//Error
IF timDissableFunctions.Q THEN 
	fbEM.bWarning := TRUE; 
	fbEM.iWarningCode := 0; 
ELSE 
	fbEM.bWarning := FALSE; 
END_IF 
IF Lynus_Standards.GVL_Energy.stNumberOfDevices.diNumberOfElectricMeters > Constants_Energy.diMaxNumberOfElectricMeters THEN 
	fbEM.bError := TRUE; 
ELSE 
	fbEM.bError := FALSE; 
END_IF
IF Lynus_Standards.GVL_Energy.stNumberOfDevices.diNumberOfElectricMeters > Constants_Energy.diMaxNumberOfElectricMeters THEN 
	fbEM.iErrorCode := 1;
ELSE 
	fbEM.iErrorCode := 0;
END_IF

timSetCounterValues(IN:= bEnable AND NOT timSetCounterValues.Q, PT:= T#2S, Q=> , ET=> );

END_FUNCTION_BLOCK

// ---- FBs/FB_EM_Beckhoff_EL3446.TcPOU
FUNCTION_BLOCK FB_EM_Beckhoff_EL3446
VAR_INPUT
	bEnable							: BOOL;											//Enable the function
  	bEnableVariantValues 			: BOOL; //Enables the Variant values to be queried using the multiplexer functions of the block
    pDpmData 						: POINTER TO ARRAY[1..20] OF UDINT;
	nSlaveAddr						: UINT;											//EtherCat Slave ID	
 	b_SubIndex						: BYTE;											//AmsNet ID Index, typically 2 or 3
 	bInvers_CH1						: BOOL;											//Invert the Output data from Channel 1 
	bInvers_CH2						: BOOL;											//Invert the Output data from Channel 2 
	bInvers_CH3						: BOOL;											//Invert the Output data from Channel 3
	bInvers_CH4						: BOOL;											//Invert the Output data from Channel 4
	bInvers_CH5						: BOOL;											//Invert the Output data from Channel 5
	bInvers_CH6						: BOOL;											//Invert the Output data from Channel 6
	uiCurrentTransformerRatio_CH1	: UINT;											//Current Transformer Ratio for Channel 1 
	uiCurrentTransformerRatio_CH2	: UINT;											//Current Transformer Ratio for Channel 2 
	uiCurrentTransformerRatio_CH3	: UINT;											//Current Transformer Ratio for Channel 3 
	uiCurrentTransformerRatio_CH4	: UINT;											//Current Transformer Ratio for Channel 4 
	uiCurrentTransformerRatio_CH5	: UINT;											//Current Transformer Ratio for Channel 5 
	uiCurrentTransformerRatio_CH6	: UINT;											//Current Transformer Ratio for Channel 6
	uiVoltagePhaseSelector_CH1		: UINT;											//Voltage Phase Selector 1/2/3 for Channel 1
	uiVoltagePhaseSelector_CH2		: UINT;											//Voltage Phase Selector 1/2/3 for Channel 2
	uiVoltagePhaseSelector_CH3		: UINT;											//Voltage Phase Selector 1/2/3 for Channel 3
	uiVoltagePhaseSelector_CH4		: UINT;											//Voltage Phase Selector 1/2/3 for Channel 4
	uiVoltagePhaseSelector_CH5		: UINT;											//Voltage Phase Selector 1/2/3 for Channel 5
	uiVoltagePhaseSelector_CH6		: UINT;											//Voltage Phase Selector 1/2/3 for Channel 6 
	bEnable3PhaseCH13				: BOOL;											//Enable 3 phase measurement Channel 1-3
	bEnable3PhaseCH46				: BOOL;											//Enable 3 phase measurement Channel 4-6
	stDataEMPowerRealTime			: ST_ElectricMeter_Output_Power;				//Output structure with Data from Electric Meter (Power Data RealTime) used adding voltage to output struct
    stEL3446_IO : MDP5001_342_066CA8C6; 
END_VAR
VAR_OUTPUT
	stDataEMPower_CH1				: ST_ElectricMeter_Output_Power;				//Output structure with Data from Electric Meter (Power Data) for Channel 1
	stDataEMCounter_CH1				: ST_ElectricMeter_Output_Counter;				//Output structure with Data from Electric Meter (Counter Data) for Channel 1
	stDataEMPowerRealTime_CH1		: ST_ElectricMeter_Output_Power;				//Output structure with Data from Electric Meter (Power Data RealTime) for Channel 1
	stDataEMCounterRealTime_CH1		: ST_ElectricMeter_Output_Counter;				//Output structure with Data from Electric Meter (Counter Data RealTime) for Channel 1

	stDataEMPower_CH2				: ST_ElectricMeter_Output_Power;				//Output structure with Data from Electric Meter (Power Data) for Channel 2
	stDataEMCounter_CH2				: ST_ElectricMeter_Output_Counter;				//Output structure with Data from Electric Meter (Counter Data) for Channel 2
	stDataEMPowerRealTime_CH2		: ST_ElectricMeter_Output_Power;				//Output structure with Data from Electric Meter (Power Data RealTime) for Channel 2
	stDataEMCounterRealTime_CH2		: ST_ElectricMeter_Output_Counter;				//Output structure with Data from Electric Meter (Counter Data RealTime) for Channel 2

	stDataEMPower_CH3				: ST_ElectricMeter_Output_Power;				//Output structure with Data from Electric Meter (Power Data) for Channel 3
	stDataEMCounter_CH3				: ST_ElectricMeter_Output_Counter;				//Output structure with Data from Electric Meter (Counter Data) for Channel 3
	stDataEMPowerRealTime_CH3		: ST_ElectricMeter_Output_Power;				//Output structure with Data from Electric Meter (Power Data RealTime) for Channel 3
	stDataEMCounterRealTime_CH3		: ST_ElectricMeter_Output_Counter;				//Output structure with Data from Electric Meter (Counter Data RealTime) for Channel 3

	stDataEMPower_CH4				: ST_ElectricMeter_Output_Power;				//Output structure with Data from Electric Meter (Power Data) for Channel 4
	stDataEMCounter_CH4				: ST_ElectricMeter_Output_Counter;				//Output structure with Data from Electric Meter (Counter Data) for Channel 4
	stDataEMPowerRealTime_CH4		: ST_ElectricMeter_Output_Power;				//Output structure with Data from Electric Meter (Power Data RealTime) for Channel 4
	stDataEMCounterRealTime_CH4		: ST_ElectricMeter_Output_Counter;				//Output structure with Data from Electric Meter (Counter Data RealTime) for Channel 4

	stDataEMPower_CH5				: ST_ElectricMeter_Output_Power;				//Output structure with Data from Electric Meter (Power Data) for Channel 5
	stDataEMCounter_CH5				: ST_ElectricMeter_Output_Counter;				//Output structure with Data from Electric Meter (Counter Data) for Channel 5
	stDataEMPowerRealTime_CH5		: ST_ElectricMeter_Output_Power;				//Output structure with Data from Electric Meter (Power Data RealTime) for Channel 5
	stDataEMCounterRealTime_CH5		: ST_ElectricMeter_Output_Counter;				//Output structure with Data from Electric Meter (Counter Data RealTime) for Channel 5

	stDataEMPower_CH6				: ST_ElectricMeter_Output_Power;				//Output structure with Data from Electric Meter (Power Data) for Channel 6
	stDataEMCounter_CH6				: ST_ElectricMeter_Output_Counter;				//Output structure with Data from Electric Meter (Counter Data) for Channel 6
	stDataEMPowerRealTime_CH6		: ST_ElectricMeter_Output_Power;				//Output structure with Data from Electric Meter (Power Data RealTime) for Channel 6
	stDataEMCounterRealTime_CH6		: ST_ElectricMeter_Output_Counter;				//Output structure with Data from Electric Meter (Counter Data RealTime) for Channel 6	
	
END_VAR
VAR
	fbEM_CH1						: FB_ElectricMeter;								//Electric Meter Function
	fbEnergyCounter_CH1				: FB_EnergyCounter;								//FB energy Counter, because the KL3403 has no nice logic for the Energy value
	fbEM_CH2						: FB_ElectricMeter;								//Electric Meter Function
	fbEnergyCounter_CH2				: FB_EnergyCounter;								//FB energy Counter, because the KL3403 has no nice logic for the Energy value
	fbEM_CH3						: FB_ElectricMeter;								//Electric Meter Function
	fbEnergyCounter_CH3				: FB_EnergyCounter;								//FB energy Counter, because the KL3403 has no nice logic for the Energy value
	fbEM_CH4						: FB_ElectricMeter;								//Electric Meter Function
	fbEnergyCounter_CH4				: FB_EnergyCounter;								//FB energy Counter, because the KL3403 has no nice logic for the Energy value
	fbEM_CH5						: FB_ElectricMeter;								//Electric Meter Function
	fbEnergyCounter_CH5				: FB_EnergyCounter;								//FB energy Counter, because the KL3403 has no nice logic for the Energy value
	fbEM_CH6						: FB_ElectricMeter;								//Electric Meter Function
	fbEnergyCounter_CH6				: FB_EnergyCounter;								//FB energy Counter, because the KL3403 has no nice logic for the Energy value
	fbEL3446_wEL3443	: FB_EL3446; 		//EL3446 | 6-channel current input terminal 1 A AC/DC for distributed power measurement (FW02 or higher) for DPM with EL3443
	
	timDissableFunctions			: TON;											//Timer to dissable the Function after Lynus_Standards.Constants_General.tTimeDissableLynusFunctions Days without connection to the Lynus Cloud
	timResetConnectionOnGVL			: TON;											//Timer to try reset the connection Flag on the GVL. (When somebody delete the Connection Function and make only a onlinechange)
	timSetCounterValues				: TON;											//Timer to set the counter values from the KL3403 Function to the EM Function
	arrPD							: ARRAY[1..7] OF FB_PersistentData_Number;		//Function to save persistent data
	byWaitInStep					: BYTE;											//Wait in Step before start to clean data on PLC
	iStateGVLData					: INT;											//State machine to handle the data on the GVL
	diCounterForGVL					: DINT;											//Counter to clean old data on GVL
	bInit: BOOL;
	m_COE_Done: BOOL;
	FB_CoE_EL3446 :FB_CoE_EL3446;
	uiVoltagePhaseSelector_old_CH1		: UINT;											
	uiVoltagePhaseSelector_old_CH2		: UINT;											
	uiVoltagePhaseSelector_old_CH3		: UINT;											
	uiVoltagePhaseSelector_old_CH4		: UINT;											
	uiVoltagePhaseSelector_old_CH5		: UINT;											
	uiVoltagePhaseSelector_old_CH6		: UINT;											
	
	f_trig_Busy: f_trig;

	real_Multiplier_CH1: REAL;
	real_Multiplier_CH2: REAL;
	real_Multiplier_CH3: REAL;
	real_Multiplier_CH4: REAL;
	real_Multiplier_CH5: REAL;
	real_Multiplier_CH6: REAL;
	

			
END_VAR

//Creator : Stefan Lackner
//Company : EfficientIO
//Date : xx.09.2023
//Version : 1.0.0.0


//With this function is possible to read out all Information from a EL3446

//NOTE for diNr.....Designation => 
//_IN = Here Data come in from other Functions or go out to other functions about the GVL
//_OUT = Here Data go out to other functions about the GVL



(*-------------------------------------------------------------Service from Backend is ready and check the connection to backen for dissabel/enable Function---------------------------------------------------------------*)

//Try to reset the variable for connection on the GVL. When all is normal then the Lynus Mqtt connection function set this variable to true in the next cycle
//When we have no connection to the backend then after Lynus_Standards.Constants_General.tTimeDissableLynusFunctions days the Function is dissabled with all of his functionalities
timResetConnectionOnGVL(IN:= NOT timResetConnectionOnGVL.Q, PT:= T#1H, Q=> , ET=> );
IF timResetConnectionOnGVL.Q THEN 
	Lynus_Standards.GVL_Communicator.bStateConnectionToEnableFunctions := FALSE; 
END_IF
IF NOT Lynus_Standards.GVL_Communicator.bStateConnectionToEnableFunctions THEN 
	timDissableFunctions.IN := TRUE; 
ELSE 
	timDissableFunctions.IN := FALSE; 
END_IF  
timDissableFunctions(IN:= , PT:= Lynus_Standards.Constants_General.tTimeDissableLynusFunctions, Q=> , ET=> );

// limit inputs
uiCurrentTransformerRatio_CH1 := LIMIT (1,uiCurrentTransformerRatio_CH1,10000);
uiCurrentTransformerRatio_CH2 := LIMIT (1,uiCurrentTransformerRatio_CH2,10000);
uiCurrentTransformerRatio_CH3 := LIMIT (1,uiCurrentTransformerRatio_CH3,10000);
uiCurrentTransformerRatio_CH4 := LIMIT (1,uiCurrentTransformerRatio_CH4,10000);
uiCurrentTransformerRatio_CH5 := LIMIT (1,uiCurrentTransformerRatio_CH5,10000);
uiCurrentTransformerRatio_CH6 := LIMIT (1,uiCurrentTransformerRatio_CH6,10000);
uiVoltagePhaseSelector_CH1 := LIMIT (1,uiVoltagePhaseSelector_CH1,3);
uiVoltagePhaseSelector_CH2 := LIMIT (1,uiVoltagePhaseSelector_CH2,3);
uiVoltagePhaseSelector_CH3 := LIMIT (1,uiVoltagePhaseSelector_CH3,3);
uiVoltagePhaseSelector_CH4 := LIMIT (1,uiVoltagePhaseSelector_CH4,3);
uiVoltagePhaseSelector_CH5 := LIMIT (1,uiVoltagePhaseSelector_CH5,3);
uiVoltagePhaseSelector_CH6 := LIMIT (1,uiVoltagePhaseSelector_CH6,3);


(*----------------------------------------------------------------------------------------EL3446 Communication----------------------------------------------------------------------------------------------*)

// write CoE values for phase selector

IF 	NOT m_COE_Done OR uiVoltagePhaseSelector_CH1 <> uiVoltagePhaseSelector_old_CH1 OR uiVoltagePhaseSelector_CH2 <> uiVoltagePhaseSelector_old_CH2 OR
 	uiVoltagePhaseSelector_CH3 <> uiVoltagePhaseSelector_old_CH3 OR uiVoltagePhaseSelector_CH4 <> uiVoltagePhaseSelector_old_CH4 OR
  	uiVoltagePhaseSelector_CH5 <> uiVoltagePhaseSelector_old_CH5 OR uiVoltagePhaseSelector_CH6 <> uiVoltagePhaseSelector_old_CH6 
	THEN
	FB_CoE_EL3446.m_start := TRUE;
	m_COE_Done := TRUE;
	 uiVoltagePhaseSelector_old_CH1 := uiVoltagePhaseSelector_CH1;
	 uiVoltagePhaseSelector_old_CH2 := uiVoltagePhaseSelector_CH2;
	 uiVoltagePhaseSelector_old_CH3 := uiVoltagePhaseSelector_CH3;
	 uiVoltagePhaseSelector_old_CH4 := uiVoltagePhaseSelector_CH4;
	 uiVoltagePhaseSelector_old_CH5 := uiVoltagePhaseSelector_CH5;
	 uiVoltagePhaseSelector_old_CH6 := uiVoltagePhaseSelector_CH6;
END_IF
f_trig_Busy(CLK := FB_CoE_EL3446.m_Busy );
IF f_trig_Busy.Q AND (FB_CoE_EL3446.m_CoE_Write_done OR FB_CoE_EL3446.m_Error) THEN 
	FB_CoE_EL3446.m_start := FALSE;
END_IF
FB_CoE_EL3446(
	m_start:= , 
	nSlaveAddr:= nSlaveAddr,
	b_SubIndex:= b_SubIndex,
	uiVoltagePhaseSelector_CH1:= uiVoltagePhaseSelector_CH1, 
	uiVoltagePhaseSelector_CH2:= uiVoltagePhaseSelector_CH2, 
	uiVoltagePhaseSelector_CH3:= uiVoltagePhaseSelector_CH3, 
	uiVoltagePhaseSelector_CH4:= uiVoltagePhaseSelector_CH4, 
	uiVoltagePhaseSelector_CH5:= uiVoltagePhaseSelector_CH5, 
	uiVoltagePhaseSelector_CH6:= uiVoltagePhaseSelector_CH6, 
	m_Busy=> , 
	m_CoE_Write_done=> , 
	udint_GetAMSNetID_Error=> , 
	udint_WriteCoE_Error=> );

fbEL3446_wEL3443(
	bEnable:= TRUE, 
	pDpmData:= pDpmData, 
	stEL3446_IO:= , 
	stStatusPhase_I1=> , 
	stStatusPhase_I2=> , 
	stStatusPhase_I3=> , 
	stStatusPhase_I4=> , 
	stStatusPhase_I5=> , 
	stStatusPhase_I6=> , 
	stDPMVariantValues=> , 
	bError=> );
fbEL3446_wEL3443.stEL3446_IO.MDP5001_342_Input := stEL3446_IO.MDP5001_342_Input;
stEL3446_IO.MDP5001_342_Output := fbEL3446_wEL3443.stEL3446_IO.MDP5001_342_Output;
//Invert the Output data, because it is possible that the current transformers have been mounted in different mounting positions.
IF NOT bInvers_CH1 THEN
	real_Multiplier_CH1 := 1;
ELSE
	real_Multiplier_CH1 := -1;
END_IF
IF NOT bInvers_CH2 THEN
	real_Multiplier_CH2 := 1;
ELSE
	real_Multiplier_CH2 := -1;
END_IF
IF NOT bInvers_CH3 THEN
	real_Multiplier_CH3 := 1;
ELSE
	real_Multiplier_CH3 := -1;
END_IF
IF NOT bInvers_CH4 THEN
	real_Multiplier_CH4 := 1;
ELSE
	real_Multiplier_CH4 := -1;
END_IF
IF NOT bInvers_CH5 THEN
	real_Multiplier_CH5 := 1;
ELSE
	real_Multiplier_CH5 := -1;
END_IF
IF NOT bInvers_CH6 THEN
	real_Multiplier_CH6 := 1;
ELSE
	real_Multiplier_CH6 := -1;
END_IF

//Function
IF NOT bEnable3PhaseCH13 THEN
	fbEM_CH1(
		bEnable:= bEnable AND NOT timDissableFunctions.Q, 
		bError:= , 
		bEnableReadOutFunction:= FALSE, 
		bWriteWithDelay:= TRUE, 
		bPowerDataInvers:= FALSE,
		bReadOutDataDone:= timSetCounterValues.Q,
		iTimeReadOutInterval:= 0, 
		iErrorCode:= , 
		iWarningCode:= , 
		lrTotalCounterEnergy_Consumption:= fbEnergyCounter_CH1.lrTotalCounterEnergy_Consumption,
		lrTotalCounterEnergy_Production:= fbEnergyCounter_CH1.lrTotalCounterEnergy_Production, 
		lrCounterEnergyT1_Consumption:= fbEnergyCounter_CH1.lrCounterEnergyT1_Consumption,
		lrCounterEnergyT2_Consumption:= fbEnergyCounter_CH1.lrCounterEnergyT2_Consumption,
		lrCounterEnergyT1_Production:= fbEnergyCounter_CH1.lrCounterEnergyT1_Production, 
		lrCounterEnergyT2_Production:= fbEnergyCounter_CH1.lrCounterEnergyT2_Production, 
		lrCurrentL1:=  fbEL3446_wEL3443.stStatusPhase_I1.fCurrent * uiCurrentTransformerRatio_CH1,
		lrVoltageL1N:= , 
		lrVoltageL1L2:= , 
		lrPowerL1:= fbEL3446_wEL3443.stStatusPhase_I1.fActive_Power * uiCurrentTransformerRatio_CH1 * real_Multiplier_CH1, 
		lrCurrentL2:= ,
		lrVoltageL2N:= , 
		lrVoltageL2L3:= , 
		lrPowerL2:= , 
		lrCurrentL3:= , 
		lrVoltageL3N:= , 
		lrVoltageL3L1:= , 
		lrPowerL3:= , 
		lrPowerTotal:= fbEM_CH1.lrPowerL1, 
		lrFrequency:= stDataEMPowerRealTime.lrFrequency,  
		lrApparentPowerTotal:= fbEL3446_wEL3443.stStatusPhase_I1.fApparent_Power * uiCurrentTransformerRatio_CH1 ,
		lrReactivePowerTotal:= fbEL3446_wEL3443.stStatusPhase_I1.fReactive_Power_Fundamental * uiCurrentTransformerRatio_CH1, 
		tTimDelayOutput:= T#5S, 
		stDataEMOutPower=> stDataEMPowerRealTime_CH1, 
		stDataEMOutPowerDelay=> stDataEMPower_CH1, 
		stDataEMOutCounter=> stDataEMCounterRealTime_CH1,
		stDataEMOutCounterDelay=> stDataEMCounter_CH1,
		bReadOutMeter=> );
	fbEM_CH2(
		bEnable:= bEnable AND NOT timDissableFunctions.Q, 
		bError:= , 
		bEnableReadOutFunction:= FALSE, 
		bWriteWithDelay:= TRUE, 
		bPowerDataInvers:= FALSE,
		bReadOutDataDone:= timSetCounterValues.Q,
		iTimeReadOutInterval:= 0, 
		iErrorCode:= , 
		iWarningCode:= , 
		lrTotalCounterEnergy_Consumption:= fbEnergyCounter_CH2.lrTotalCounterEnergy_Consumption,
		lrTotalCounterEnergy_Production:= fbEnergyCounter_CH2.lrTotalCounterEnergy_Production, 
		lrCounterEnergyT1_Consumption:= fbEnergyCounter_CH2.lrCounterEnergyT1_Consumption,
		lrCounterEnergyT2_Consumption:= fbEnergyCounter_CH2.lrCounterEnergyT2_Consumption,
		lrCounterEnergyT1_Production:= fbEnergyCounter_CH2.lrCounterEnergyT1_Production, 
		lrCounterEnergyT2_Production:= fbEnergyCounter_CH2.lrCounterEnergyT2_Production, 
		lrCurrentL1:=  fbEL3446_wEL3443.stStatusPhase_I2.fCurrent * uiCurrentTransformerRatio_CH2,
		lrVoltageL1N:= , 
		lrVoltageL1L2:= , 
		lrPowerL1:= fbEL3446_wEL3443.stStatusPhase_I2.fActive_Power * uiCurrentTransformerRatio_CH2 * real_Multiplier_CH2, 
		lrCurrentL2:= ,
		lrVoltageL2N:= , 
		lrVoltageL2L3:= , 
		lrPowerL2:= , 
		lrCurrentL3:= , 
		lrVoltageL3N:= , 
		lrVoltageL3L1:= , 
		lrPowerL3:= , 
		lrPowerTotal:= fbEM_CH2.lrPowerL1, 
		lrFrequency:= stDataEMPowerRealTime.lrFrequency, 
		lrApparentPowerTotal:= fbEL3446_wEL3443.stStatusPhase_I2.fApparent_Power * uiCurrentTransformerRatio_CH2 ,
		lrReactivePowerTotal:= fbEL3446_wEL3443.stStatusPhase_I2.fReactive_Power_Fundamental * uiCurrentTransformerRatio_CH2, 
		tTimDelayOutput:= T#5S, 
		stDataEMOutPower=> stDataEMPowerRealTime_CH2, 
		stDataEMOutPowerDelay=> stDataEMPower_CH2, 
		stDataEMOutCounter=> stDataEMCounterRealTime_CH2,
		stDataEMOutCounterDelay=> stDataEMCounter_CH2,
		bReadOutMeter=> );
	fbEM_CH3(
		bEnable:= bEnable AND NOT timDissableFunctions.Q, 
		bError:= , 
		bEnableReadOutFunction:= FALSE, 
		bWriteWithDelay:= TRUE, 
		bPowerDataInvers:= FALSE,
		bReadOutDataDone:= timSetCounterValues.Q,
		iTimeReadOutInterval:= 0, 
		iErrorCode:= , 
		iWarningCode:= , 
		lrTotalCounterEnergy_Consumption:= fbEnergyCounter_CH3.lrTotalCounterEnergy_Consumption,
		lrTotalCounterEnergy_Production:= fbEnergyCounter_CH3.lrTotalCounterEnergy_Production, 
		lrCounterEnergyT1_Consumption:= fbEnergyCounter_CH3.lrCounterEnergyT1_Consumption,
		lrCounterEnergyT2_Consumption:= fbEnergyCounter_CH3.lrCounterEnergyT2_Consumption,
		lrCounterEnergyT1_Production:= fbEnergyCounter_CH3.lrCounterEnergyT1_Production, 
		lrCounterEnergyT2_Production:= fbEnergyCounter_CH3.lrCounterEnergyT2_Production, 
		lrCurrentL1:=  fbEL3446_wEL3443.stStatusPhase_I3.fCurrent * uiCurrentTransformerRatio_CH3,
		lrVoltageL1N:= , 
		lrVoltageL1L2:= , 
		lrPowerL1:= fbEL3446_wEL3443.stStatusPhase_I3.fActive_Power * uiCurrentTransformerRatio_CH3 * real_Multiplier_CH3, 
		lrCurrentL2:= ,
		lrVoltageL2N:= , 
		lrVoltageL2L3:= , 
		lrPowerL2:= , 
		lrCurrentL3:= , 
		lrVoltageL3N:= , 
		lrVoltageL3L1:= , 
		lrPowerL3:= , 
		lrPowerTotal:= fbEM_CH3.lrPowerL1, 
		lrFrequency:= stDataEMPowerRealTime.lrFrequency,
		lrApparentPowerTotal:= fbEL3446_wEL3443.stStatusPhase_I3.fApparent_Power * uiCurrentTransformerRatio_CH3 ,
		lrReactivePowerTotal:= fbEL3446_wEL3443.stStatusPhase_I3.fReactive_Power_Fundamental * uiCurrentTransformerRatio_CH3, 
		tTimDelayOutput:= T#5S, 
		stDataEMOutPower=> stDataEMPowerRealTime_CH3, 
		stDataEMOutPowerDelay=> stDataEMPower_CH3, 
		stDataEMOutCounter=> stDataEMCounterRealTime_CH3,
		stDataEMOutCounterDelay=> stDataEMCounter_CH3,
		bReadOutMeter=> );
	fbEnergyCounter_CH1(
		byActiveTariff:= 1, 
		lrPowerInput:= (fbEM_CH1.lrPowerL1) / 1000, 
		lrTotalCounterEnergy_Consumption=> , 
		lrTotalCounterEnergy_Production=> , 
		lrCounterEnergyT1_Consumption=> , 
		lrCounterEnergyT2_Consumption=> , 
		lrCounterEnergyT1_Production=> , 
		lrCounterEnergyT2_Production=> );
	fbEnergyCounter_CH2(
		byActiveTariff:= 1, 
		lrPowerInput:= (fbEM_CH2.lrPowerL1) / 1000, 
		lrTotalCounterEnergy_Consumption=> , 
		lrTotalCounterEnergy_Production=> , 
		lrCounterEnergyT1_Consumption=> , 
		lrCounterEnergyT2_Consumption=> , 
		lrCounterEnergyT1_Production=> , 
		lrCounterEnergyT2_Production=> );
	fbEnergyCounter_CH3(
		byActiveTariff:= 1, 
		lrPowerInput:= (fbEM_CH3.lrPowerL1) / 1000, 
		lrTotalCounterEnergy_Consumption=> , 
		lrTotalCounterEnergy_Production=> , 
		lrCounterEnergyT1_Consumption=> , 
		lrCounterEnergyT2_Consumption=> , 
		lrCounterEnergyT1_Production=> , 
		lrCounterEnergyT2_Production=> );
	CASE uiVoltagePhaseSelector_CH1 OF
		1: 	fbEM_CH1.lrVoltageL1N := stDataEMPowerRealTime.lrVoltageL1N;
		2: 	fbEM_CH1.lrVoltageL1N := stDataEMPowerRealTime.lrVoltageL2N;
		3: 	fbEM_CH1.lrVoltageL1N := stDataEMPowerRealTime.lrVoltageL3N;	
	END_CASE
	CASE uiVoltagePhaseSelector_CH2 OF
		1: 	fbEM_CH2.lrVoltageL1N := stDataEMPowerRealTime.lrVoltageL1N;
		2: 	fbEM_CH2.lrVoltageL1N := stDataEMPowerRealTime.lrVoltageL2N;
		3: 	fbEM_CH2.lrVoltageL1N := stDataEMPowerRealTime.lrVoltageL3N;	
	END_CASE
	CASE uiVoltagePhaseSelector_CH3 OF
		1: 	fbEM_CH3.lrVoltageL1N := stDataEMPowerRealTime.lrVoltageL1N;
		2: 	fbEM_CH3.lrVoltageL1N := stDataEMPowerRealTime.lrVoltageL2N;
		3: 	fbEM_CH3.lrVoltageL1N := stDataEMPowerRealTime.lrVoltageL3N;	
	END_CASE	
ELSE
	fbEM_CH1(
		bEnable:= bEnable AND NOT timDissableFunctions.Q, 
		bError:= , 
		bEnableReadOutFunction:= FALSE, 
		bWriteWithDelay:= TRUE, 
		bPowerDataInvers:= FALSE,
		bReadOutDataDone:= timSetCounterValues.Q,
		iTimeReadOutInterval:= 0, 
		iErrorCode:= , 
		iWarningCode:= , 
		lrTotalCounterEnergy_Consumption:= fbEnergyCounter_CH1.lrTotalCounterEnergy_Consumption,
		lrTotalCounterEnergy_Production:= fbEnergyCounter_CH1.lrTotalCounterEnergy_Production, 
		lrCounterEnergyT1_Consumption:= fbEnergyCounter_CH1.lrCounterEnergyT1_Consumption,
		lrCounterEnergyT2_Consumption:= fbEnergyCounter_CH1.lrCounterEnergyT2_Consumption,
		lrCounterEnergyT1_Production:= fbEnergyCounter_CH1.lrCounterEnergyT1_Production, 
		lrCounterEnergyT2_Production:= fbEnergyCounter_CH1.lrCounterEnergyT2_Production, 
		lrCurrentL1:=  fbEL3446_wEL3443.stStatusPhase_I1.fCurrent * uiCurrentTransformerRatio_CH1,
		lrVoltageL1N:= stDataEMPowerRealTime.lrVoltageL1N, 
		lrVoltageL1L2:= stDataEMPowerRealTime.lrVoltageL1L2, 
		lrPowerL1:= fbEL3446_wEL3443.stStatusPhase_I1.fActive_Power * uiCurrentTransformerRatio_CH1 * real_Multiplier_CH1, 
		lrCurrentL2:= fbEL3446_wEL3443.stStatusPhase_I2.fCurrent * uiCurrentTransformerRatio_CH2,
		lrVoltageL2N:= stDataEMPowerRealTime.lrVoltageL2N, 
		lrVoltageL2L3:=stDataEMPowerRealTime.lrVoltageL2L3 , 
		lrPowerL2:= fbEL3446_wEL3443.stStatusPhase_I2.fActive_Power * uiCurrentTransformerRatio_CH2 * real_Multiplier_CH2, 
		lrCurrentL3:=  fbEL3446_wEL3443.stStatusPhase_I3.fCurrent * uiCurrentTransformerRatio_CH3, 
		lrVoltageL3N:= stDataEMPowerRealTime.lrVoltageL3N, 
		lrVoltageL3L1:= stDataEMPowerRealTime.lrVoltageL3L1 , 
		lrPowerL3:= fbEL3446_wEL3443.stStatusPhase_I3.fActive_Power * uiCurrentTransformerRatio_CH3 * real_Multiplier_CH3, 
		lrPowerTotal:= fbEM_CH1.lrPowerL1 + fbEM_CH1.lrPowerL2 + fbEM_CH1.lrPowerL3,
		lrFrequency:= stDataEMPowerRealTime.lrFrequency, 
		lrApparentPowerTotal:= fbEL3446_wEL3443.stStatusPhase_I1.fApparent_Power * uiCurrentTransformerRatio_CH1 + fbEL3446_wEL3443.stStatusPhase_I2.fApparent_Power * uiCurrentTransformerRatio_CH2 + fbEL3446_wEL3443.stStatusPhase_I3.fApparent_Power * uiCurrentTransformerRatio_CH3,
		lrReactivePowerTotal:= fbEL3446_wEL3443.stStatusPhase_I1.fReactive_Power_Fundamental * uiCurrentTransformerRatio_CH1 + fbEL3446_wEL3443.stStatusPhase_I2.fReactive_Power_Fundamental * uiCurrentTransformerRatio_CH2 + fbEL3446_wEL3443.stStatusPhase_I3.fReactive_Power_Fundamental * uiCurrentTransformerRatio_CH3, 
		tTimDelayOutput:= T#5S, 
		stDataEMOutPower=> stDataEMPowerRealTime_CH1, 
		stDataEMOutPowerDelay=> stDataEMPower_CH1, 
		stDataEMOutCounter=> stDataEMCounterRealTime_CH1,
		stDataEMOutCounterDelay=> stDataEMCounter_CH1,
		bReadOutMeter=> );	
	fbEnergyCounter_CH1(
		byActiveTariff:= 1, 
		lrPowerInput:= (fbEM_CH1.lrPowerTotal) / 1000, 
		lrTotalCounterEnergy_Consumption=> , 
		lrTotalCounterEnergy_Production=> , 
		lrCounterEnergyT1_Consumption=> , 
		lrCounterEnergyT2_Consumption=> , 
		lrCounterEnergyT1_Production=> , 
		lrCounterEnergyT2_Production=> );
END_IF	
IF NOT bEnable3PhaseCH46 THEN 	
	fbEM_CH4(
		bEnable:= bEnable AND NOT timDissableFunctions.Q, 
		bError:= , 
		bEnableReadOutFunction:= FALSE, 
		bWriteWithDelay:= TRUE, 
		bPowerDataInvers:= FALSE,
		bReadOutDataDone:= timSetCounterValues.Q,
		iTimeReadOutInterval:= 0, 
		iErrorCode:= , 
		iWarningCode:= , 
		lrTotalCounterEnergy_Consumption:= fbEnergyCounter_CH4.lrTotalCounterEnergy_Consumption,
		lrTotalCounterEnergy_Production:= fbEnergyCounter_CH4.lrTotalCounterEnergy_Production, 
		lrCounterEnergyT1_Consumption:= fbEnergyCounter_CH4.lrCounterEnergyT1_Consumption,
		lrCounterEnergyT2_Consumption:= fbEnergyCounter_CH4.lrCounterEnergyT2_Consumption,
		lrCounterEnergyT1_Production:= fbEnergyCounter_CH4.lrCounterEnergyT1_Production, 
		lrCounterEnergyT2_Production:= fbEnergyCounter_CH4.lrCounterEnergyT2_Production, 
		lrCurrentL1:=  fbEL3446_wEL3443.stStatusPhase_I4.fCurrent * uiCurrentTransformerRatio_CH4,
		lrVoltageL1N:= , 
		lrVoltageL1L2:= , 
		lrPowerL1:= fbEL3446_wEL3443.stStatusPhase_I4.fActive_Power * uiCurrentTransformerRatio_CH4 * real_Multiplier_CH4, 
		lrCurrentL2:= ,
		lrVoltageL2N:= , 
		lrVoltageL2L3:= , 
		lrPowerL2:= , 
		lrCurrentL3:= , 
		lrVoltageL3N:= , 
		lrVoltageL3L1:= , 
		lrPowerL3:= , 
		lrPowerTotal:= fbEM_CH4.lrPowerL1, 
		lrFrequency:= stDataEMPowerRealTime.lrFrequency,
		lrApparentPowerTotal:= fbEL3446_wEL3443.stStatusPhase_I4.fApparent_Power * uiCurrentTransformerRatio_CH4 ,
		lrReactivePowerTotal:= fbEL3446_wEL3443.stStatusPhase_I4.fReactive_Power_Fundamental * uiCurrentTransformerRatio_CH4, 
		tTimDelayOutput:= T#5S, 
		stDataEMOutPower=> stDataEMPowerRealTime_CH4, 
		stDataEMOutPowerDelay=> stDataEMPower_CH4, 
		stDataEMOutCounter=> stDataEMCounterRealTime_CH4,
		stDataEMOutCounterDelay=> stDataEMCounter_CH4,
		bReadOutMeter=> );
	fbEM_CH5(
		bEnable:= bEnable AND NOT timDissableFunctions.Q, 
		bError:= , 
		bEnableReadOutFunction:= FALSE, 
		bWriteWithDelay:= TRUE, 
		bPowerDataInvers:= FALSE,
		bReadOutDataDone:= timSetCounterValues.Q,
		iTimeReadOutInterval:= 0, 
		iErrorCode:= , 
		iWarningCode:= , 
		lrTotalCounterEnergy_Consumption:= fbEnergyCounter_CH5.lrTotalCounterEnergy_Consumption,
		lrTotalCounterEnergy_Production:= fbEnergyCounter_CH5.lrTotalCounterEnergy_Production, 
		lrCounterEnergyT1_Consumption:= fbEnergyCounter_CH5.lrCounterEnergyT1_Consumption,
		lrCounterEnergyT2_Consumption:= fbEnergyCounter_CH5.lrCounterEnergyT2_Consumption,
		lrCounterEnergyT1_Production:= fbEnergyCounter_CH5.lrCounterEnergyT1_Production, 
		lrCounterEnergyT2_Production:= fbEnergyCounter_CH5.lrCounterEnergyT2_Production, 
		lrCurrentL1:=  fbEL3446_wEL3443.stStatusPhase_I5.fCurrent * uiCurrentTransformerRatio_CH5,
		lrVoltageL1N:= , 
		lrVoltageL1L2:= , 
		lrPowerL1:= fbEL3446_wEL3443.stStatusPhase_I5.fActive_Power * uiCurrentTransformerRatio_CH5 * real_Multiplier_CH5, 
		lrCurrentL2:= ,
		lrVoltageL2N:= , 
		lrVoltageL2L3:= , 
		lrPowerL2:= , 
		lrCurrentL3:= , 
		lrVoltageL3N:= , 
		lrVoltageL3L1:= , 
		lrPowerL3:= , 
		lrPowerTotal:= fbEM_CH5.lrPowerL1, 
		lrFrequency:= stDataEMPowerRealTime.lrFrequency,
		lrApparentPowerTotal:= fbEL3446_wEL3443.stStatusPhase_I5.fApparent_Power * uiCurrentTransformerRatio_CH5 ,
		lrReactivePowerTotal:= fbEL3446_wEL3443.stStatusPhase_I5.fReactive_Power_Fundamental * uiCurrentTransformerRatio_CH5, 
		tTimDelayOutput:= T#5S, 
		stDataEMOutPower=> stDataEMPowerRealTime_CH5, 
		stDataEMOutPowerDelay=> stDataEMPower_CH5, 
		stDataEMOutCounter=> stDataEMCounterRealTime_CH5,
		stDataEMOutCounterDelay=> stDataEMCounter_CH5,
		bReadOutMeter=> );
	fbEM_CH6(
		bEnable:= bEnable AND NOT timDissableFunctions.Q, 
		bError:= , 
		bEnableReadOutFunction:= FALSE, 
		bWriteWithDelay:= TRUE, 
		bPowerDataInvers:= FALSE,
		bReadOutDataDone:= timSetCounterValues.Q,
		iTimeReadOutInterval:= 0, 
		iErrorCode:= , 
		iWarningCode:= , 
		lrTotalCounterEnergy_Consumption:= fbEnergyCounter_CH6.lrTotalCounterEnergy_Consumption,
		lrTotalCounterEnergy_Production:= fbEnergyCounter_CH6.lrTotalCounterEnergy_Production, 
		lrCounterEnergyT1_Consumption:= fbEnergyCounter_CH6.lrCounterEnergyT1_Consumption,
		lrCounterEnergyT2_Consumption:= fbEnergyCounter_CH6.lrCounterEnergyT2_Consumption,
		lrCounterEnergyT1_Production:= fbEnergyCounter_CH6.lrCounterEnergyT1_Production, 
		lrCounterEnergyT2_Production:= fbEnergyCounter_CH6.lrCounterEnergyT2_Production, 
		lrCurrentL1:=  fbEL3446_wEL3443.stStatusPhase_I6.fCurrent * uiCurrentTransformerRatio_CH6,
		lrVoltageL1N:= , 
		lrVoltageL1L2:= , 
		lrPowerL1:= fbEL3446_wEL3443.stStatusPhase_I6.fActive_Power * uiCurrentTransformerRatio_CH6 * real_Multiplier_CH6, 
		lrCurrentL2:= ,
		lrVoltageL2N:= , 
		lrVoltageL2L3:= , 
		lrPowerL2:= , 
		lrCurrentL3:= , 
		lrVoltageL3N:= , 
		lrVoltageL3L1:= , 
		lrPowerL3:= , 
		lrPowerTotal:= fbEM_CH6.lrPowerL1, 
		lrFrequency:= stDataEMPowerRealTime.lrFrequency,
		lrApparentPowerTotal:= fbEL3446_wEL3443.stStatusPhase_I6.fApparent_Power * uiCurrentTransformerRatio_CH6 ,
		lrReactivePowerTotal:= fbEL3446_wEL3443.stStatusPhase_I6.fReactive_Power_Fundamental * uiCurrentTransformerRatio_CH6, 
		tTimDelayOutput:= T#5S, 
		stDataEMOutPower=> stDataEMPowerRealTime_CH6, 
		stDataEMOutPowerDelay=> stDataEMPower_CH6, 
		stDataEMOutCounter=> stDataEMCounterRealTime_CH6,
		stDataEMOutCounterDelay=> stDataEMCounter_CH6,
		bReadOutMeter=> );
	fbEnergyCounter_CH4(
		byActiveTariff:= 1, 
		lrPowerInput:= (fbEM_CH4.lrPowerL1) / 1000, 
		lrTotalCounterEnergy_Consumption=> , 
		lrTotalCounterEnergy_Production=> , 
		lrCounterEnergyT1_Consumption=> , 
		lrCounterEnergyT2_Consumption=> , 
		lrCounterEnergyT1_Production=> , 
		lrCounterEnergyT2_Production=> );
	fbEnergyCounter_CH5(
		byActiveTariff:= 1, 
		lrPowerInput:= (fbEM_CH5.lrPowerL1) / 1000, 
		lrTotalCounterEnergy_Consumption=> , 
		lrTotalCounterEnergy_Production=> , 
		lrCounterEnergyT1_Consumption=> , 
		lrCounterEnergyT2_Consumption=> , 
		lrCounterEnergyT1_Production=> , 
		lrCounterEnergyT2_Production=> );
	fbEnergyCounter_CH6(
		byActiveTariff:= 1, 
		lrPowerInput:= (fbEM_CH6.lrPowerL1) / 1000, 
		lrTotalCounterEnergy_Consumption=> , 
		lrTotalCounterEnergy_Production=> , 
		lrCounterEnergyT1_Consumption=> , 
		lrCounterEnergyT2_Consumption=> , 
		lrCounterEnergyT1_Production=> , 
		lrCounterEnergyT2_Production=> );
	CASE uiVoltagePhaseSelector_CH4 OF
		1: 	fbEM_CH4.lrVoltageL1N := stDataEMPowerRealTime.lrVoltageL1N;
		2: 	fbEM_CH4.lrVoltageL1N := stDataEMPowerRealTime.lrVoltageL2N;
		3: 	fbEM_CH4.lrVoltageL1N := stDataEMPowerRealTime.lrVoltageL3N;	
	END_CASE
	CASE uiVoltagePhaseSelector_CH5 OF
		1: 	fbEM_CH5.lrVoltageL1N := stDataEMPowerRealTime.lrVoltageL1N;
		2: 	fbEM_CH5.lrVoltageL1N := stDataEMPowerRealTime.lrVoltageL2N;
		3: 	fbEM_CH5.lrVoltageL1N := stDataEMPowerRealTime.lrVoltageL3N;	
	END_CASE
	CASE uiVoltagePhaseSelector_CH6 OF
		1: 	fbEM_CH6.lrVoltageL1N := stDataEMPowerRealTime.lrVoltageL1N;
		2: 	fbEM_CH6.lrVoltageL1N := stDataEMPowerRealTime.lrVoltageL2N;
		3: 	fbEM_CH6.lrVoltageL1N := stDataEMPowerRealTime.lrVoltageL3N;	
	END_CASE
ELSE 
	fbEM_CH4(
		bEnable:= bEnable AND NOT timDissableFunctions.Q, 
		bError:= , 
		bEnableReadOutFunction:= FALSE, 
		bWriteWithDelay:= TRUE, 
		bPowerDataInvers:= FALSE,
		bReadOutDataDone:= timSetCounterValues.Q,
		iTimeReadOutInterval:= 0, 
		iErrorCode:= , 
		iWarningCode:= , 
		lrTotalCounterEnergy_Consumption:= fbEnergyCounter_CH4.lrTotalCounterEnergy_Consumption,
		lrTotalCounterEnergy_Production:= fbEnergyCounter_CH4.lrTotalCounterEnergy_Production, 
		lrCounterEnergyT1_Consumption:= fbEnergyCounter_CH4.lrCounterEnergyT1_Consumption,
		lrCounterEnergyT2_Consumption:= fbEnergyCounter_CH4.lrCounterEnergyT2_Consumption,
		lrCounterEnergyT1_Production:= fbEnergyCounter_CH4.lrCounterEnergyT1_Production, 
		lrCounterEnergyT2_Production:= fbEnergyCounter_CH4.lrCounterEnergyT2_Production, 
		lrCurrentL1:=  fbEL3446_wEL3443.stStatusPhase_I4.fCurrent * uiCurrentTransformerRatio_CH4,
		lrVoltageL1N:= stDataEMPowerRealTime.lrVoltageL1N, 
		lrVoltageL1L2:= stDataEMPowerRealTime.lrVoltageL1L2, 
		lrPowerL1:= fbEL3446_wEL3443.stStatusPhase_I4.fActive_Power * uiCurrentTransformerRatio_CH4 * real_Multiplier_CH4, 
		lrCurrentL2:= fbEL3446_wEL3443.stStatusPhase_I5.fCurrent * uiCurrentTransformerRatio_CH5,
		lrVoltageL2N:= stDataEMPowerRealTime.lrVoltageL2N, 
		lrVoltageL2L3:=stDataEMPowerRealTime.lrVoltageL2L3 , 
		lrPowerL2:= fbEL3446_wEL3443.stStatusPhase_I5.fActive_Power * uiCurrentTransformerRatio_CH5 * real_Multiplier_CH5, 
		lrCurrentL3:=  fbEL3446_wEL3443.stStatusPhase_I6.fCurrent * uiCurrentTransformerRatio_CH6, 
		lrVoltageL3N:= stDataEMPowerRealTime.lrVoltageL3N, 
		lrVoltageL3L1:= stDataEMPowerRealTime.lrVoltageL3L1 , 
		lrPowerL3:= fbEL3446_wEL3443.stStatusPhase_I6.fActive_Power * uiCurrentTransformerRatio_CH6 * real_Multiplier_CH6, 
		lrPowerTotal:= fbEM_CH4.lrPowerL1 + fbEM_CH4.lrPowerL2 + fbEM_CH4.lrPowerL3,
		lrFrequency:= stDataEMPowerRealTime.lrFrequency, 
		lrApparentPowerTotal:= fbEL3446_wEL3443.stStatusPhase_I4.fApparent_Power * uiCurrentTransformerRatio_CH4 + fbEL3446_wEL3443.stStatusPhase_I5.fApparent_Power * uiCurrentTransformerRatio_CH5 + fbEL3446_wEL3443.stStatusPhase_I6.fApparent_Power * uiCurrentTransformerRatio_CH6,
		lrReactivePowerTotal:= fbEL3446_wEL3443.stStatusPhase_I4.fReactive_Power_Fundamental * uiCurrentTransformerRatio_CH4 + fbEL3446_wEL3443.stStatusPhase_I5.fReactive_Power_Fundamental * uiCurrentTransformerRatio_CH5 + fbEL3446_wEL3443.stStatusPhase_I6.fReactive_Power_Fundamental * uiCurrentTransformerRatio_CH6, 
		tTimDelayOutput:= T#5S, 
		stDataEMOutPower=> stDataEMPowerRealTime_CH4, 
		stDataEMOutPowerDelay=> stDataEMPower_CH4, 
		stDataEMOutCounter=> stDataEMCounterRealTime_CH4,
		stDataEMOutCounterDelay=> stDataEMCounter_CH4,
		bReadOutMeter=> );	
	fbEnergyCounter_CH4(
		byActiveTariff:= 1, 
		lrPowerInput:= (fbEM_CH4.lrPowerTotal) / 1000, 
		lrTotalCounterEnergy_Consumption=> , 
		lrTotalCounterEnergy_Production=> , 
		lrCounterEnergyT1_Consumption=> , 
		lrCounterEnergyT2_Consumption=> , 
		lrCounterEnergyT1_Production=> , 
		lrCounterEnergyT2_Production=> );
END_IF
(*----------------------------------------------------------------------------------------Electric Meter Function----------------------------------------------------------------------------------------------*)

//Error
IF timDissableFunctions.Q THEN 
	fbEM_CH1.bWarning := TRUE; 
	fbEM_CH1.iWarningCode := 0; 
ELSE 
	fbEM_CH1.bWarning := FALSE; 
END_IF 
IF Lynus_Standards.GVL_Energy.stNumberOfDevices.diNumberOfElectricMeters > Constants_Energy.diMaxNumberOfElectricMeters THEN 
	fbEM_CH1.bError := TRUE; 
ELSE 
	fbEM_CH1.bError := FALSE; 
END_IF
IF Lynus_Standards.GVL_Energy.stNumberOfDevices.diNumberOfElectricMeters > Constants_Energy.diMaxNumberOfElectricMeters THEN 
	fbEM_CH1.iErrorCode := 1;
ELSE 
	fbEM_CH1.iErrorCode := 0;
END_IF

timSetCounterValues(IN:= bEnable AND NOT timSetCounterValues.Q, PT:= T#2S, Q=> , ET=> );

END_FUNCTION_BLOCK

// ---- FBs/FB_CoE_EL3446.TcPOU
FUNCTION_BLOCK FB_CoE_EL3446
VAR_INPUT
	m_start: BOOL;
	nSlaveAddr	:UINT;
	b_SubIndex	:BYTE;
	uiVoltagePhaseSelector_CH1		: UINT;											//Voltage Phase Selector 1/2/3 for Channel 1
	uiVoltagePhaseSelector_CH2		: UINT;											//Voltage Phase Selector 1/2/3 for Channel 2
	uiVoltagePhaseSelector_CH3		: UINT;											//Voltage Phase Selector 1/2/3 for Channel 3
	uiVoltagePhaseSelector_CH4		: UINT;											//Voltage Phase Selector 1/2/3 for Channel 4
	uiVoltagePhaseSelector_CH5		: UINT;											//Voltage Phase Selector 1/2/3 for Channel 5
	uiVoltagePhaseSelector_CH6		: UINT;											//Voltage Phase Selector 1/2/3 for Channel 6 
END_VAR
VAR_OUTPUT
	m_Busy: BOOL;
	m_CoE_Write_done: BOOL;
	m_Error: bool;
	udint_GetAMSNetID_Error: UDINT;
	udint_WriteCoE_Error: UDINT;
END_VAR
VAR
	i_State	:UINT:=1;
	fb_GetAMSNetID	:FB_GetLocalAmsNetId;
  	fb_coe_write          : FB_EcCoESdoWrite; // Function Block for writing in CoE


	r_trig_Start: R_trig;
	i_errorCount: INT;
	i_AMSNetID_ReadOut_Succesfull: INT;
	str_AMSNetID: STRING(30);
 	nValue     : UdINT ; (* variable to be written to the CoE Object *)
 	
	i_CoE_Write_Succesfull: INT;
	udint_Value: UDINT;
	real_Value: REAL;

END_VAR


r_trig_Start(Clk := m_start);
b_SubIndex := LIMIT (1,b_SubIndex,8);
CASE i_State OF
	1: 		// wait for start
	IF r_trig_Start.Q THEN
		i_State := i_State+1;
		m_CoE_Write_done := FALSE;
		m_Busy := TRUE;
		m_Error := FALSE;
	END_IF

	2:		// read out ams net ID	
	fb_GetAMSNetID.bExecute := TRUE;
	i_State := i_State+1;
	
	3: 		// wait for read ot
	IF fb_GetAMSNetID.bBusy = FALSE AND NOT fb_GetAMSNetID.bError = TRUE THEN
		fb_GetAMSNetID.bExecute := FALSE;
		i_AMSNetID_ReadOut_Succesfull := i_AMSNetID_ReadOut_Succesfull+1;
		i_State := i_State+1;
	ELSIF fb_GetAMSNetID.bError = TRUE THEN
		fb_GetAMSNetID.bExecute := FALSE;
		i_State := 100;
	END_IF
	
	4: 		// read out AMS Net ID done, convert received data
	str_AMSNetID := concat(BYTE_TO_STRING(fb_GetAMSNetID.AddrBytes[0]),'.');
	str_AMSNetID := concat(str_AMSNetID,BYTE_TO_STRING(fb_GetAMSNetID.AddrBytes[1]));
	str_AMSNetID := concat(str_AMSNetID,'.');	
	str_AMSNetID := concat(str_AMSNetID,BYTE_TO_STRING(fb_GetAMSNetID.AddrBytes[2]));
	str_AMSNetID := concat(str_AMSNetID,'.');
	str_AMSNetID := concat(str_AMSNetID,BYTE_TO_STRING(fb_GetAMSNetID.AddrBytes[3]));
	str_AMSNetID := concat(str_AMSNetID,'.');
	str_AMSNetID := concat(str_AMSNetID,BYTE_TO_STRING(b_SubIndex));
	str_AMSNetID := concat(str_AMSNetID,'.1');
	
	i_State := 10;

	10: 	// write channel 1 phase Selector
	fb_coe_write.bExecute 	:= TRUE;
	fb_coe_write.nIndex		:= 16#8000;
	fb_coe_write.nSubIndex	:= 16#11; 
	udint_Value 			:= UINT_TO_UDINT(uiVoltagePhaseSelector_CH1);
	fb_coe_write.pSrcBuf	:= ADR(udint_Value);
	fb_coe_write.cbBufLen	:= SIZEOF(udint_Value);
	i_State := i_State+1;
	
	11: 	// wait for done or error
	IF NOT fb_coe_write.bBusy AND NOT fb_coe_write.bError THEN
		fb_coe_write.bExecute 	:= FALSE;
		i_CoE_Write_Succesfull := i_CoE_Write_Succesfull+1;
		i_State := i_State+1;
	ELSIF fb_coe_write.bError THEN
		fb_coe_write.bExecute 	:= FALSE;
		i_State := 100;
	END_IF

	12:		// wait 
	i_State := 20;
	
	20: 	// write channel 2 phase Selector
	fb_coe_write.bExecute 	:= TRUE;
	fb_coe_write.nIndex		:= 16#8010;
	fb_coe_write.nSubIndex	:= 16#11; 
	udint_Value 			:= UINT_TO_UDINT(uiVoltagePhaseSelector_CH2);
	fb_coe_write.pSrcBuf	:= ADR(udint_Value);
	fb_coe_write.cbBufLen	:= SIZEOF(udint_Value);
	i_State := i_State+1;
	
	21: 	// wait for done or error
	IF NOT fb_coe_write.bBusy AND NOT fb_coe_write.bError THEN
		fb_coe_write.bExecute 	:= FALSE;
		i_CoE_Write_Succesfull := i_CoE_Write_Succesfull+1;
		i_State := i_State+1;
	ELSIF fb_coe_write.bError THEN
		fb_coe_write.bExecute 	:= FALSE;
		i_State := 100;
	END_IF

	22:		// wait 
	i_State := 30;

	30: 	// write channel 3 phase Selector
	fb_coe_write.bExecute 	:= TRUE;
	fb_coe_write.nIndex		:= 16#8020;
	fb_coe_write.nSubIndex	:= 16#11; 
	udint_Value 			:= UINT_TO_UDINT(uiVoltagePhaseSelector_CH3);
	fb_coe_write.pSrcBuf	:= ADR(udint_Value);
	fb_coe_write.cbBufLen	:= SIZEOF(udint_Value);
	i_State := i_State+1;
	
	31: 	// wait for done or error
	IF NOT fb_coe_write.bBusy AND NOT fb_coe_write.bError THEN
		fb_coe_write.bExecute 	:= FALSE;
		i_CoE_Write_Succesfull := i_CoE_Write_Succesfull+1;
		i_State := i_State+1;
	ELSIF fb_coe_write.bError THEN
		fb_coe_write.bExecute 	:= FALSE;
		i_State := 100;
	END_IF

	32:		// wait 
	i_State := 40;
	
	40: 	// write channel 4 phase Selector
	fb_coe_write.bExecute 	:= TRUE;
	fb_coe_write.nIndex		:= 16#8030;
	fb_coe_write.nSubIndex	:= 16#11; 
	udint_Value 			:= UINT_TO_UDINT(uiVoltagePhaseSelector_CH4);
	fb_coe_write.pSrcBuf	:= ADR(udint_Value);
	fb_coe_write.cbBufLen	:= SIZEOF(udint_Value);
	i_State := i_State+1;
	
	41: 	// wait for done or error
	IF NOT fb_coe_write.bBusy AND NOT fb_coe_write.bError THEN
		fb_coe_write.bExecute 	:= FALSE;
		i_CoE_Write_Succesfull := i_CoE_Write_Succesfull+1;
		i_State := i_State+1;
	ELSIF fb_coe_write.bError THEN
		fb_coe_write.bExecute 	:= FALSE;
		i_State := 100;
	END_IF

	42:		// wait 
	i_State := 50;		

	50: 	// write channel 5 phase Selector
	fb_coe_write.bExecute 	:= TRUE;
	fb_coe_write.nIndex		:= 16#8040;
	fb_coe_write.nSubIndex	:= 16#11; 
	udint_Value 			:= UINT_TO_UDINT(uiVoltagePhaseSelector_CH5);
	fb_coe_write.pSrcBuf	:= ADR(udint_Value);
	fb_coe_write.cbBufLen	:= SIZEOF(udint_Value);
	i_State := i_State+1;
	
	51: 	// wait for done or error
	IF NOT fb_coe_write.bBusy AND NOT fb_coe_write.bError THEN
		fb_coe_write.bExecute 	:= FALSE;
		i_CoE_Write_Succesfull := i_CoE_Write_Succesfull+1;
		i_State := i_State+1;
	ELSIF fb_coe_write.bError THEN
		fb_coe_write.bExecute 	:= FALSE;
		i_State := 100;
	END_IF

	52:		// wait 
	i_State := 60;		

	60: 	// write channel 6 phase Selector
	fb_coe_write.bExecute 	:= TRUE;
	fb_coe_write.nIndex		:= 16#8050;
	fb_coe_write.nSubIndex	:= 16#11; 
	udint_Value 			:= UINT_TO_UDINT(uiVoltagePhaseSelector_CH6);
	fb_coe_write.pSrcBuf	:= ADR(udint_Value);
	fb_coe_write.cbBufLen	:= SIZEOF(udint_Value);
	i_State := i_State+1;
	
	61: 	// wait for done or error
	IF NOT fb_coe_write.bBusy AND NOT fb_coe_write.bError THEN
		fb_coe_write.bExecute 	:= FALSE;
		i_CoE_Write_Succesfull := i_CoE_Write_Succesfull+1;
		i_State := i_State+1;
	ELSIF fb_coe_write.bError THEN
		fb_coe_write.bExecute 	:= FALSE;
		i_State := 100;
	END_IF

	62:		// wait 
	m_CoE_Write_done := TRUE;
	m_Busy := FALSE;
	i_State := 1;		
	
	100: 	//error state
	i_errorCount := i_errorCount +1;
	udint_GetAMSNetID_Error := fb_GetAMSNetID.nErrId;
	udint_WriteCoE_Error := fb_coe_write.nErrId;
	m_Busy := FALSE;
	m_Error := true;
	i_State := 1;

END_CASE


fb_GetAMSNetID(
	bExecute:= , 
	tTimeOut:= T#2S, 
	bBusy=> , 
	bError=> , 
	nErrId=> , 
	AddrString=> , 
	AddrBytes=> );
	
fb_coe_write(
	sNetId:= str_AMSNetID, 
	nSlaveAddr:= nSlaveAddr, 
	nSubIndex:= , 
	nIndex:= , 
    pSrcBuf    := ,
    cbBufLen   := ,
	bExecute:= , 
	tTimeout:= T#2S , 
	bBusy=> , 
	bError=> , 
	nErrId=> );

END_FUNCTION_BLOCK

// ---- FBs/FB_ModBus_100Registers_FC3_inclID.TcPOU
FUNCTION_BLOCK FB_ModBus_100Registers_FC3_inclID
VAR_INPUT PERSISTENT
	m_Enable					: BOOL;						//Enable the Fuctionblock and his logic
	str_IPAdress				: STRING(15);				//IP Adress of the meter
	w_Adress					: WORD;						//modbus adress
	usint_Quantity				: usINT;						//Number of Words to get polled, max 100
	usint_ID					: USINT;						//Number of Words to get polled, max 100
END_VAR
VAR_OUTPUT
	m_PollSuccessful			: BOOL;						//Poll succesfull		
	w_Array_Received			: ARRAY[1..100] OF WORD;	// received data
	udint_Error_ID				: UDINT;					// ERR ID FB_MBReadRegs
END_VAR
VAR
	
	timer_Delay					: TON;						//Timer for Delay between Requests
	
	timer_DelayStart			: TON;						//Timer to start the state machine with Delay after enabling or after the system ist restartet
	
	timer_TimeOut				: TON;						//Timer for Timeout MB Read
	
	iStateModbusRead			: INT;						//State machine for read out Data over Modbus RTU
	
	fbMBRead_FC3				: FB_MBReadRegs  ;		//Modbus Read Function (FC3)
	
	ftrig_PEnable				: f_trig;					//Internal positive Edge
	
	iStateModbusError			: INT;						//State machine for error out Data over Modbus TCP/IP	
	
	FPError_FC_3				: R_TRIG;					//Internal positive Edge
	
	arrBuffer_FC3				: ARRAY[1..100] OF WORD;		//Buffer with Data from FC3
	
	timer_Connection_ok			: TON;
	int_Data_Received			: INT;
	
	m_MBTCPError				: BOOL;
	
	int_Data_Received_old		: INT;
	
	timer_Connection_ok_TOF	: TOF;
	
	fbConvertWordToDword		: FB_CV_WORD_TO_DWORD;			//Convert Word to Dword
	
	m_Poll_ok: BOOL;
	
	timer_Wait: Ton;
	int_TimeoutError: INT;
	int_FC3Error: INT;

END_VAR

(*	{attribute 'hide'}--------------------------------------------------------------------------------------------Limits-------------------------------------------------------------------------------------*)

w_Adress := LIMIT(0,w_Adress,60000);
usint_Quantity := LIMIT(1,usint_Quantity,100);
	
(*--------------------------------------------------------------------------------------------State Machine Read--------------------------------------------------------------------------------------*)

//Timer for Delay
timer_Delay(IN:= , PT:= T#50MS, Q=> , ET=> );

//Timeout Timer is dissabled when the Init Step is aktiv or the function is not enabled
IF iStateModbusRead = 0 OR NOT m_Enable THEN 
	timer_Timeout.IN := FALSE; 
END_IF
timer_Timeout(IN:= , PT:= T#1S, Q=> , ET=> );

//Enable with Delay that not all sockets have to be created at the same time
timer_DelayStart(IN:= m_Enable, PT:= T#1S, Q=> , ET=> );
ftrig_PEnable(CLK:= timer_DelayStart.Q, Q=> );

IF ftrig_PEnable.Q AND iStateModbusRead = 0 THEN 
	iStateModbusRead := 1; 
END_IF		
IF usint_ID < 1 OR usint_ID >255 THEN 
	usint_ID := 1;
END_IF		
//Not Enabled
IF NOT m_Enable THEN 
	iStateModbusRead := 0; 
	iStateModbusError := 0; 
END_IF		
		
CASE iStateModbusRead OF

	0://Init Step 
		timer_Delay.IN := FALSE;
		fbMBRead_FC3.bExecute := FALSE;
		m_Poll_ok:=FALSE;
		int_Data_Received:=0;
	
		iStateModbusRead := 1;
	
	1://read the required registers
		//Start Read
		fbMBRead_FC3.nQuantity := usint_Quantity;
		fbMBRead_FC3.nMBAddr := w_Adress;
		fbMBRead_FC3.bExecute := TRUE;
		fbMBRead_FC3.nUnitID := usint_ID;
		timer_Timeout.IN := TRUE;
		IF fbMBRead_FC3.bBusy THEN 
			timer_Delay.IN := TRUE; 
		END_IF
		
		//Wait for Delay, copy Data and then next step
		IF NOT fbMBRead_FC3.bBusy AND NOT fbMBRead_FC3.bError AND timer_Delay.Q THEN
			m_Poll_ok:=TRUE;
			int_Data_Received:=int_Data_Received+1;
			m_MBTCPError := FALSE; 
			
			w_Array_Received := arrBuffer_FC3;
			
			
			//Go to Next Step
			timer_Timeout.IN := FALSE;
			fbMBRead_FC3.bExecute := FALSE;
			timer_Delay.IN := FALSE;		
			iStateModbusRead := 3;
		END_IF	

		//Error or Timeout
		IF FPError_FC_3.Q THEN 
			iStateModbusError := 300;
			int_FC3Error := int_FC3Error+1;
		ELSIF timer_Timeout.Q THEN  
			timer_Timeout.IN := FALSE; 	
			iStateModbusError := 300;
			int_TimeoutError := int_TimeoutError+1;
		END_IF
		
	
	3://Wait and go to step 1
		//1 because 0 is the Init Step for Read
		timer_Wait.IN := TRUE;
		
		IF timer_Wait.Q = TRUE THEN
			iStateModbusRead := 1;
			timer_Wait.IN :=FALSE;
		END_IF

			
		
		//Error on Master, changes on Inputs or Timeout
		IF timer_Timeout.Q THEN 
			iStateModbusError := 300; 
		END_IF
	
END_CASE

(* wait timer*)

timer_Wait(PT:=T#3S);


(*------------------------------------------------------------------Error and Warning----------------------------------------------------------------------------*)	
 
timer_Connection_ok			(In:=int_Data_Received<>int_Data_Received_old,PT:=T#10S);
timer_Connection_ok_TOF		(In:=NOT(int_Data_Received<>int_Data_Received_old) AND int_Data_Received>3 ,PT:=T#20S);
int_Data_Received_old:=int_Data_Received;
m_PollSuccessful:=NOT timer_Connection_ok.Q AND timer_Connection_ok_TOF.Q ;

(*------------------------------------------------------------------------------------------Modbus TCP Functions---------------------------------------------------------------------------------------------*)

fbMBRead_FC3(	sIPAddr:= str_IPAdress, 
				nTCPPort:= 502,
				cbLength:= SIZEOF(arrBuffer_FC3), 
				pDestAddr:= ADR(arrBuffer_FC3), 
				tTimeout:= T#10S,
				nErrId => udint_Error_ID);

FPError_FC_3(CLK:= fbMBRead_FC3.bError, Q=> );		

(*------------------------------------------------------------------------------------------State Machine Error---------------------------------------------------------------------------------------------*)	

CASE iStateModbusError OF
	
	300://Error
		timer_Wait.IN :=TRUE;
		timer_Delay.IN := FALSE;
		fbMBRead_FC3.bExecute := FALSE;
		m_MBTCPError := TRUE; 		
		m_Poll_ok:=FALSE;
		int_Data_Received:=0;
				//Restart from new with the Read out part after an Error
		IF timer_Wait.Q = TRUE THEN
			iStateModbusRead := 0;	
			iStateModbusError := 0;
			timer_Wait.IN :=FALSE;
			timer_Timeout.IN := FALSE;
		END_IF		
							
END_CASE

END_FUNCTION_BLOCK

// ---- POUs/prgPV.TcPOU
PROGRAM prgPV
VAR
	fbPV1_1					: FB_Symo_PV_Inverter_int_1_DM_30_Inverter_1;
	fbPV1_2					: FB_Symo_PV_Inverter_INT_1_DM_30_Inverter_1;
	lrPowerPV				: LREAL;				//{#lynus.ag#()}
	lrPowerPV_1				: LREAL;				//{#lynus.ag#()}
	lrPowerPV_2				: LREAL;				//{#lynus.ag#()}
	lrPowerPV_3				: LREAL;				//{#lynus.ag#()}
	lrPowerPV_4				: LREAL;				//{#lynus.ag#()}
	lrPowerPV_5				: LREAL;				//{#lynus.ag#()}
	lrPowerPV_6				: LREAL;				//{#lynus.ag#()}
	lrPowerPV_7				: LREAL;				//{#lynus.ag#()}
	lrPowerPV_8				: LREAL;				//{#lynus.ag#()}

	fbCounterPV_1			: FB_EnergyCounter;
	fbCounterPV_2			: FB_EnergyCounter;
	fbCounterPV_3			: FB_EnergyCounter;
	fbCounterPV_4			: FB_EnergyCounter;
	fbCounterPV_5			: FB_EnergyCounter;
	fbCounterPV_6			: FB_EnergyCounter;
	fbCounterPV_7			: FB_EnergyCounter;
	fbCounterPV_8			: FB_EnergyCounter;


	fbCounterPV_total			: FB_EnergyCounter;

END_VAR
VAR PERSISTENT
	lrCounterPV_1	: LREAL;						//{#lynus.ag#()}
	lrCounterPV_2	: LREAL;						//{#lynus.ag#()}
	lrCounterPV_3	: LREAL;						//{#lynus.ag#()}
	lrCounterPV_4	: LREAL;						//{#lynus.ag#()}
	lrCounterPV_5	: LREAL;						//{#lynus.ag#()}
	lrCounterPV_6	: LREAL;						//{#lynus.ag#()}
	lrCounterPV_7	: LREAL;						//{#lynus.ag#()}
	lrCounterPV_8	: LREAL;						//{#lynus.ag#()}
	lrCounterPV		: LREAL;						//{#lynus.ag#()}
END_VAR




fbPV1_1(
	bEnable:= TRUE, 
	sIPAdress:= '192.168.1.130', 
	arrUnitID_Inverter:= , 
	arrDataSymo10=> , 
	stDataEMPower_PV=> , 
	stDataEMCounter_PV=> , 
	diNrOfEM_OUT_PV=> );
fbPV1_1.arrUnitID_Inverter[1] := 6;
fbPV1_1.arrUnitID_Inverter[2] := 7;
fbPV1_1.arrUnitID_Inverter[3] := 8;


fbPV1_2(
	bEnable:= TRUE, 
	sIPAdress:= '192.168.1.131', 
	arrUnitID_Inverter:= , 
	arrDataSymo10=> , 
	stDataEMPower_PV=> , 
	stDataEMCounter_PV=> , 
	diNrOfEM_OUT_PV=> );
fbPV1_2.arrUnitID_Inverter[1] := 1;
fbPV1_2.arrUnitID_Inverter[2] := 2;
fbPV1_2.arrUnitID_Inverter[3] := 3;
fbPV1_2.arrUnitID_Inverter[4] := 4;
fbPV1_2.arrUnitID_Inverter[5] := 5;

lrPowerPV_1 := fbPV1_2.arrDataSymo10[1].lrPowerAcInverter;
lrPowerPV_2 := fbPV1_2.arrDataSymo10[2].lrPowerAcInverter;
lrPowerPV_3 := fbPV1_2.arrDataSymo10[3].lrPowerAcInverter;
lrPowerPV_4 := fbPV1_2.arrDataSymo10[4].lrPowerAcInverter;
lrPowerPV_5 := fbPV1_2.arrDataSymo10[5].lrPowerAcInverter;
lrPowerPV_6 := fbPV1_1.arrDataSymo10[1].lrPowerAcInverter;
lrPowerPV_7 := fbPV1_1.arrDataSymo10[2].lrPowerAcInverter;
lrPowerPV_8 := fbPV1_1.arrDataSymo10[3].lrPowerAcInverter;
	


lrPowerPV := lrPowerPV_1 + lrPowerPV_2 + lrPowerPV_3 + lrPowerPV_4 + lrPowerPV_5 + lrPowerPV_6 + lrPowerPV_7 + lrPowerPV_8;


// kWh Counters

fbCounterPV_1(
	byActiveTariff:= 1, 
	lrPowerInput:= lrPowerPV_1, 
	lrTotalCounterEnergy_Consumption=> , 
	lrTotalCounterEnergy_Production=> , 
	lrCounterEnergyT1_Consumption=> , 
	lrCounterEnergyT2_Consumption=> , 
	lrCounterEnergyT1_Production=> , 
	lrCounterEnergyT2_Production=> );
	
IF fbCounterPV_1.lrTotalCounterEnergy_Consumption > lrCounterPV_1 THEN  	
	lrCounterPV_1 := fbCounterPV_1.lrTotalCounterEnergy_Consumption;
END_IF

fbCounterPV_2(
	byActiveTariff:= 1, 
	lrPowerInput:= lrPowerPV_2, 
	lrTotalCounterEnergy_Consumption=> , 
	lrTotalCounterEnergy_Production=> , 
	lrCounterEnergyT1_Consumption=> , 
	lrCounterEnergyT2_Consumption=> , 
	lrCounterEnergyT1_Production=> , 
	lrCounterEnergyT2_Production=> );
	
IF fbCounterPV_2.lrTotalCounterEnergy_Consumption > lrCounterPV_2 THEN  	
	lrCounterPV_2 := fbCounterPV_2.lrTotalCounterEnergy_Consumption;
END_IF

fbCounterPV_3(
	byActiveTariff:= 1, 
	lrPowerInput:= lrPowerPV_3, 
	lrTotalCounterEnergy_Consumption=> , 
	lrTotalCounterEnergy_Production=> , 
	lrCounterEnergyT1_Consumption=> , 
	lrCounterEnergyT2_Consumption=> , 
	lrCounterEnergyT1_Production=> , 
	lrCounterEnergyT2_Production=> );
	
IF fbCounterPV_3.lrTotalCounterEnergy_Consumption > lrCounterPV_3 THEN  	
	lrCounterPV_3 := fbCounterPV_3.lrTotalCounterEnergy_Consumption;
END_IF

fbCounterPV_4(
	byActiveTariff:= 1, 
	lrPowerInput:= lrPowerPV_4, 
	lrTotalCounterEnergy_Consumption=> , 
	lrTotalCounterEnergy_Production=> , 
	lrCounterEnergyT1_Consumption=> , 
	lrCounterEnergyT2_Consumption=> , 
	lrCounterEnergyT1_Production=> , 
	lrCounterEnergyT2_Production=> );
	
IF fbCounterPV_4.lrTotalCounterEnergy_Consumption > lrCounterPV_4 THEN  	
	lrCounterPV_4 := fbCounterPV_4.lrTotalCounterEnergy_Consumption;
END_IF

fbCounterPV_5(
	byActiveTariff:= 1, 
	lrPowerInput:= lrPowerPV_5, 
	lrTotalCounterEnergy_Consumption=> , 
	lrTotalCounterEnergy_Production=> , 
	lrCounterEnergyT1_Consumption=> , 
	lrCounterEnergyT2_Consumption=> , 
	lrCounterEnergyT1_Production=> , 
	lrCounterEnergyT2_Production=> );
	
IF fbCounterPV_5.lrTotalCounterEnergy_Consumption > lrCounterPV_5 THEN  	
	lrCounterPV_5 := fbCounterPV_5.lrTotalCounterEnergy_Consumption;
END_IF

fbCounterPV_6(
	byActiveTariff:= 1, 
	lrPowerInput:= lrPowerPV_6, 
	lrTotalCounterEnergy_Consumption=> , 
	lrTotalCounterEnergy_Production=> , 
	lrCounterEnergyT1_Consumption=> , 
	lrCounterEnergyT2_Consumption=> , 
	lrCounterEnergyT1_Production=> , 
	lrCounterEnergyT2_Production=> );
	
IF fbCounterPV_6.lrTotalCounterEnergy_Consumption > lrCounterPV_6 THEN  	
	lrCounterPV_6 := fbCounterPV_6.lrTotalCounterEnergy_Consumption;
END_IF

fbCounterPV_7(
	byActiveTariff:= 1, 
	lrPowerInput:= lrPowerPV_7, 
	lrTotalCounterEnergy_Consumption=> , 
	lrTotalCounterEnergy_Production=> , 
	lrCounterEnergyT1_Consumption=> , 
	lrCounterEnergyT2_Consumption=> , 
	lrCounterEnergyT1_Production=> , 
	lrCounterEnergyT2_Production=> );
	
IF fbCounterPV_7.lrTotalCounterEnergy_Consumption > lrCounterPV_7 THEN  	
	lrCounterPV_7 := fbCounterPV_7.lrTotalCounterEnergy_Consumption;
END_IF

fbCounterPV_8(
	byActiveTariff:= 1, 
	lrPowerInput:= lrPowerPV_8, 
	lrTotalCounterEnergy_Consumption=> , 
	lrTotalCounterEnergy_Production=> , 
	lrCounterEnergyT1_Consumption=> , 
	lrCounterEnergyT2_Consumption=> , 
	lrCounterEnergyT1_Production=> , 
	lrCounterEnergyT2_Production=> );
	
IF fbCounterPV_8.lrTotalCounterEnergy_Consumption > lrCounterPV_8 THEN  	
	lrCounterPV_8 := fbCounterPV_8.lrTotalCounterEnergy_Consumption;
END_IF

fbCounterPV_total(
	byActiveTariff:= 1, 
	lrPowerInput:= lrPowerPV, 
	lrTotalCounterEnergy_Consumption=> , 
	lrTotalCounterEnergy_Production=> , 
	lrCounterEnergyT1_Consumption=> , 
	lrCounterEnergyT2_Consumption=> , 
	lrCounterEnergyT1_Production=> , 
	lrCounterEnergyT2_Production=> );
	
IF fbCounterPV_total.lrTotalCounterEnergy_Consumption > lrCounterPV THEN  	
	lrCounterPV := fbCounterPV_total.lrTotalCounterEnergy_Consumption;
END_IF

END_PROGRAM

// ---- FBs/FB_Symo_PV_Inverter_INT_1_DM_30_Inverter_1.TcPOU
{attribute 'hide_all_locals'}
FUNCTION_BLOCK FB_Symo_PV_Inverter_INT_1_DM_30_Inverter_1
VAR_INPUT PERSISTENT
	bEnable						: BOOL;												//True = Function is enabled, FALSE = Function is dissabled, no new Data
	sIPAdress					: STRING(15);										//IP Adress from the Inverter
	arrUnitID_Inverter			: ARRAY[1..30] OF BYTE;								//Array with the Unit ID's from each Inverter (Max 30 Inverters) (ID = 1 to 247) (0 = No Inverter)
END_VAR
VAR_OUTPUT
	arrDataSymo10				: ARRAY[1..30] OF ST_Symo_PV_OutData;				//Output structure with Data from Symo 10
	stDataEMPower_PV			: ST_ElectricMeter_Output_Power;					//Output structure with Data from Electric Meter PV (Power Data)
	stDataEMCounter_PV			: ST_ElectricMeter_Output_Counter;					//Output structure with Data from Electric Meter PV (Counter Data)
	diNrOfEM_OUT_PV				: DINT;												//Active Number from the Electric Meter for using on other functions
END_VAR
VAR
	fbElMeter					: FB_ElectricMeter;									//Electric Meter Function 
	fbNumberDevice				: FB_NumberOfDevice;								//Function block to calcualte the number of the Device
	fbConvertEnergyRegister		: FB_CV_WORD_TO_UDINT;								//Convert function
	fbMBRead_FC3				: FB_MBReadRegs;									//Modbus Read Function (FC3)
	timDelay					: TON;												//Timer for Delay between Requests
	timTimeout					: TON;												//Timer for Timeout
	timDissableFunctions		: TON;												//Timer to dissable the Function after Lynus_Standards.Constants_General.tTimeDissableLynusFunctions Days without connection to the Lynus Cloud
	timResetConnectionOnGVL		: TON;												//Timer to try reset the connection Flag on the GVL. (When somebody delete the Connection Function and make only a onlinechange)
	FPEnable					: R_TRIG;											//Internal positive Edge
	FPError_FC_3				: R_TRIG;											//Internal positive Edge
	PD_String					: FB_PersistentData_String;							//Function to save persistent data
	arrUnitID_Inverter_CP		: ARRAY[1..30] OF BYTE; 							//Array with unit IDs to compare it when we have a change on the Inputs
	arrBuffer_FC3				: ARRAY[1..37] OF WORD;								//Buffer with Data from FC3
	arrCurrentL1				: ARRAY[1..30] OF LREAL;							//Array with the Current from L1 from each Inverter
	arrCurrentL2				: ARRAY[1..30] OF LREAL;							//Array with the Current from L2 from each Inverter
	arrCurrentL3				: ARRAY[1..30] OF LREAL;							//Array with the Current from L3 from each Inverter
	arrVoltageL1L2				: ARRAY[1..30] OF LREAL;							//Array with the Voltage from L1-L2 from each Inverter
	arrVoltageL2L3				: ARRAY[1..30] OF LREAL;							//Array with the Voltage from L2-L3 from each Inverter
	arrVoltageL3L1				: ARRAY[1..30] OF LREAL;							//Array with the Voltage from L3-L1 from each Inverter
	arrVoltageL1N				: ARRAY[1..30] OF LREAL;							//Array with the Voltage from L1-N from each Inverter
	arrVoltageL2N				: ARRAY[1..30] OF LREAL;							//Array with the Voltage from L2-N from each Inverter
	arrVoltageL3N				: ARRAY[1..30] OF LREAL;							//Array with the Voltage from L3-N from each Inverter
	arrACPower					: ARRAY[1..30] OF LREAL;							//Array with the AC Power from each Inverter
	arrFrequency				: ARRAY[1..30] OF LREAL;							//Array with the Frequency from each Inverter
	arrApparentPower			: ARRAY[1..30] OF LREAL;							//Array with the Apparent Power from each Inverter
	arrReactivePower			: ARRAY[1..30] OF LREAL;							//Array with the Reactive Power from each Inverter
	arrProductionEnergy			: ARRAY[1..30] OF LREAL;							//Array with the Production Energy from each Inverter
	arrPD						: ARRAY[1..31] OF FB_PersistentData_Number;			//Function to save persistent data 
	bErrorDevice				: BOOL;												//When 1 or more Inverters has a Error, then thsi Flag is true
	byInverterInProgress		: BYTE;												//Shows what Inverter is at the moment in Progress in the State machine to read out the data
	byTotalInverter				: BYTE;												//Summ of total Inverters. (Depends on the unit IDs that are not 0.) 
	byLPForInverter				: BYTE; 											//Variable for Loop to calculate some things for the Inverters
	byWaitInStep				: BYTE;												//Wait in Step before start to clean data on PLC
	iStateGVLData				: INT;												//State machine to handle the data on the GVL
	iStateModbus				: INT;												//State variable for Statemachine
	iStateModbus_CP				: INT;												//Compare State variable
	diCounterForGVL				: DINT;												//Counter to clean old data on GVL
	rValBefWToOut				: REAL;												//Value to check the received data from the inverter befor wirte to the output structure
	lrCheckValue				: LREAL;											//Internal Value to check the value before convert
	lrCounterEnergyProduction	: LREAL;											//Check counter state before write new one
END_VAR

//Creator : Kai Ebensperger
//Company : Lynus AG
//Date : 01.09.2021
//Version : 1.0.0.0

//With this function its possible to read out values from the Symo PV Inverter from the factory Fronius
//This Function read out the Values from 1 Fronius Datamanager with maximal 30 Inverter.
//The protocol to the Inverter is Modbus TCP
//Versions that are supported : 1.1.5-0
//Attention. To access the registers, an offset of 1 must always be subtracted. Register 40001 would then be on register 40000.
//This Function use the INT+Scalfactor Format
//You can query the register data of the individual devices using the Modbus device ID (UnitID).
//Each inverter has its own number stored on the display under "Setup" -> "Datcom"-> "Inverter number".
//Inverter number 00 = Modbus ID 100
//Inverter number 01 = Modbus ID 01
//Inverter number 02 = Modbus ID 02 etc.
//Internal in the GVL this function is 1 PV Plant. We display the summ ov all values from each Inverter

//Changes about AC power
//Date : 29.03.2020
//Version : 1.1.0.0

//NOTE for diNr.....Designation => 
//_IN = Here Data come in from other Functions or go out to other functions about the GVL
//_OUT = Here Data go out to other functions about the GVL

(*------------------------------------------------------------------------------------------General Input Part---------------------------------------------------------------------------------------------*)

//Check limitation
FOR byLPForInverter := 1 TO 30 BY 1 DO
	arrUnitID_Inverter[byLPForInverter] := LIMIT(0,arrUnitID_Inverter[byLPForInverter],247);
END_FOR

(*-------------------------------------------------------------Calcualte the number of EM System---------------------------------------------------------------*)

fbNumberDevice(
	diActualNumberOfDevices:= Lynus_Standards.GVL_Energy.stNumberOfDevices.diNumberOfElectricMeters, 
	diMaxNumberOfDevices:= Constants_Energy.diMaxNumberOfElectricMeters, 
	udiCounterOnlineChange:= TwinCAT_SystemInfoVarList._AppInfo.OnlineChangeCnt, 
	bNumberIsCalculatet=> , 
	bFPNumberIsCalculatet=> , 
	bOnlineChange=> , 
	diNumberForThisDevice=> diNrOfEM_OUT_PV, 
	diNumberOfTotalDevices=> );

//Write new Numer on GVL
IF fbNumberDevice.bFPNumberIsCalculatet THEN
	Lynus_Standards.GVL_Energy.stNumberOfDevices.diNumberOfElectricMeters := fbNumberDevice.diNumberOfTotalDevices;	
END_IF 

//Delete old Number on GVL
IF fbNumberDevice.bOnlineChange THEN 
	Lynus_Standards.GVL_Energy.stNumberOfDevices.diNumberOfElectricMeters := diNrOfEM_OUT_PV;	
		iStateGVLData := 1; 
END_IF

(*-------------------------------------------------------------Service from Backend is ready and check the connection to backen for dissabel/enable Function---------------------------------------------------------------*)

//Try to reset the variable for connection on the GVL. When all is normal then the Lynus Mqtt connection function set this variable to true in the next cycle
//When we have no connection to the backend then after Lynus_Standards.Constants_General.tTimeDissableLynusFunctions days the Function is dissabled with all of his functionalities
timResetConnectionOnGVL(IN:= NOT timResetConnectionOnGVL.Q, PT:= T#1H, Q=> , ET=> );
	IF timResetConnectionOnGVL.Q THEN Lynus_Standards.GVL_Communicator.bStateConnectionToEnableFunctions := FALSE; END_IF
		IF NOT Lynus_Standards.GVL_Communicator.bStateConnectionToEnableFunctions THEN timDissableFunctions.IN := TRUE; ELSE timDissableFunctions.IN := FALSE; END_IF  
			timDissableFunctions(IN:= , PT:= Lynus_Standards.Constants_General.tTimeDissableLynusFunctions, Q=> , ET=> );

(*------------------------------------------------------------------------------------------Calcualte the Max Number of Inverters---------------------------------------------------------------------------------------------*)
	
byTotalInverter := 0;
	FOR byLPForInverter := 1 TO 30 BY 1 DO
		IF arrUnitID_Inverter[byLPForInverter] <> 0 THEN byTotalInverter := byTotalInverter + 1; END_IF 
	END_FOR	
	
(*------------------------------------------------------------------------------------------State Machine---------------------------------------------------------------------------------------------*)

//Enable
FPEnable(CLK:= bEnable, Q=> );
	IF FPEnable.Q AND iStateModbus = 0 AND byTotalInverter > 0 THEN iStateModbus := 1; END_IF
		IF NOT bEnable OR timDissableFunctions.Q OR byTotalInverter = 0 OR MEMCMP(ADR(arrUnitID_Inverter),ADR(arrUnitID_Inverter_CP),SIZEOF(arrUnitID_Inverter_CP)) <> 0 THEN iStateModbus := 0; END_IF

//Timer for delay
timDelay(IN:= , PT:= T#50MS, Q=> , ET=> );	

//Timer for Timeout in Statemachine
	IF iStateModbus = iStateModbus_CP THEN timTimeout.IN := TRUE; ELSE timTimeout.IN := FALSE; END_IF
		IF iStateModbus = 0 THEN timTimeout.IN := FALSE; END_IF
timTimeout(IN:= , PT:= T#20S, Q=> , ET=> );	

//Statemachine
CASE iStateModbus OF
	
	0://Init Step
		iStateModbus_CP := iStateModbus;
			timDelay.IN := FALSE;
		
		FOR byLPForInverter := 1 TO 30 BY 1 DO 
			arrDataSymo10[byLPForInverter].bFunctionIsActive := FALSE;
				arrDataSymo10[byLPForInverter].eOperatingStateInverter := E_Symo_PV_OperatingState.eNoDataReceived;
					arrDataSymo10[byLPForInverter].lrPowerAcInverter := 0;
			arrCurrentL1[byLPForInverter] := 0;
				arrCurrentL2[byLPForInverter] := 0;
			arrCurrentL3[byLPForInverter] := 0;
				arrVoltageL1L2[byLPForInverter] := 0;
			arrVoltageL2L3[byLPForInverter] := 0;
				arrVoltageL3L1[byLPForInverter] := 0;
			arrVoltageL1N[byLPForInverter] := 0;
				arrVoltageL2N[byLPForInverter] := 0;
			arrVoltageL3N[byLPForInverter] := 0;
				arrACPower[byLPForInverter] := 0;
			arrFrequency[byLPForInverter] := 0;
				arrApparentPower[byLPForInverter] := 0;
			arrReactivePower[byLPForInverter] := 0;
				arrProductionEnergy[byLPForInverter] := 0;
		END_FOR	
				fbMBRead_FC3.bExecute := FALSE;
					lrCheckValue := 0;
						rValBefWToOut := 0;
						
		//After reset the Arrays when we have a change on the Unit ID's we restart the State Machine
		IF MEMCMP(ADR(arrUnitID_Inverter),ADR(arrUnitID_Inverter_CP),SIZEOF(arrUnitID_Inverter_CP)) <> 0 AND bEnable AND byTotalInverter > 0 THEN
			iStateModbus := 1;
				arrUnitID_Inverter_CP := arrUnitID_Inverter;
		END_IF	 
		
	1://Search the Unit ID to read out the Data for each Inverter with Unit ID <> 0
		iStateModbus_CP := iStateModbus;
		
		IF byInverterInProgress >= 30 THEN byInverterInProgress := 0; END_IF
		
		byInverterInProgress := byInverterInProgress + 1;
			byInverterInProgress := LIMIT(1,byInverterInProgress,30);	
		
		IF arrUnitID_Inverter[byInverterInProgress] <> 0 THEN iStateModbus := 2; END_IF
								
	2://Read out first Registers from 40072 to 40108
		arrDataSymo10[byInverterInProgress].bFunctionIsActive := TRUE;
			iStateModbus_CP := iStateModbus;
		
		fbMBRead_FC3.nQuantity := 37;
			fbMBRead_FC3.nMBAddr := 40071;
				fbMBRead_FC3.bExecute := TRUE;
					fbMBRead_FC3.nUnitID := arrUnitID_Inverter[byInverterInProgress];
			
		IF fbMBRead_FC3.bBusy THEN timDelay.IN := TRUE; END_IF
		
		//Wait for Delay, copy Data and then next step
		IF NOT fbMBRead_FC3.bBusy AND NOT fbMBRead_FC3.bError AND timDelay.Q AND WORD_TO_INT(arrBuffer_FC3[5]) >= -10 AND WORD_TO_INT(arrBuffer_FC3[5]) <= 10 AND WORD_TO_INT(arrBuffer_FC3[12]) >= -10 AND WORD_TO_INT(arrBuffer_FC3[12]) <= 10 AND
			WORD_TO_INT(arrBuffer_FC3[14]) >= -10 AND WORD_TO_INT(arrBuffer_FC3[14]) <= 10 AND WORD_TO_INT(arrBuffer_FC3[16]) >= -10 AND WORD_TO_INT(arrBuffer_FC3[16]) <= 10 AND WORD_TO_INT(arrBuffer_FC3[18]) >= -10 AND WORD_TO_INT(arrBuffer_FC3[18]) <= 10 AND
				WORD_TO_INT(arrBuffer_FC3[20]) >= -10 AND WORD_TO_INT(arrBuffer_FC3[20]) <= 10 AND WORD_TO_INT(arrBuffer_FC3[25]) >= -10 AND WORD_TO_INT(arrBuffer_FC3[25]) <= 10 THEN
					//Copy Data Current L1
					rValBefWToOut := WORD_TO_REAL(arrBuffer_FC3[2]);
						lrCheckValue := rValBefWToOut * EXPT(10,WORD_TO_INT(arrBuffer_FC3[5]));	
							IF lrCheckValue >= - 3.402823E+38 AND lrCheckValue <= 3.402823E+38 THEN 
								arrCurrentL1[byInverterInProgress] := lrCheckValue;
							ELSE
								iStateModbus := 300;
									arrDataSymo10[byInverterInProgress].eErrorState := E_Symo_PV_Error.eSymo10TooBigValueReceived;		
							END_IF
					//Copy Data Current L2
					rValBefWToOut := WORD_TO_REAL(arrBuffer_FC3[3]);
						lrCheckValue := rValBefWToOut * EXPT(10,WORD_TO_INT(arrBuffer_FC3[5]));	
							IF lrCheckValue >= - 3.402823E+38 AND lrCheckValue <= 3.402823E+38 THEN 
								arrCurrentL2[byInverterInProgress] := lrCheckValue;
							ELSE
								iStateModbus := 300;
									arrDataSymo10[byInverterInProgress].eErrorState := E_Symo_PV_Error.eSymo10TooBigValueReceived;		
							END_IF
					//Copy Data Current L3
					rValBefWToOut := WORD_TO_REAL(arrBuffer_FC3[4]);
						lrCheckValue := rValBefWToOut * EXPT(10,WORD_TO_INT(arrBuffer_FC3[5]));	
							IF lrCheckValue >= - 3.402823E+38 AND lrCheckValue <= 3.402823E+38 THEN 
								arrCurrentL3[byInverterInProgress] := lrCheckValue;
							ELSE
								iStateModbus := 300;
									arrDataSymo10[byInverterInProgress].eErrorState := E_Symo_PV_Error.eSymo10TooBigValueReceived;		
							END_IF
					//Copy Data Voltage L1-L2
					rValBefWToOut := WORD_TO_REAL(arrBuffer_FC3[6]);
						lrCheckValue := rValBefWToOut * EXPT(10,WORD_TO_INT(arrBuffer_FC3[12]));	
							IF lrCheckValue >= - 3.402823E+38 AND lrCheckValue <= 3.402823E+38 THEN 
								arrVoltageL1L2[byInverterInProgress] := lrCheckValue;
							ELSE
								iStateModbus := 300;
									arrDataSymo10[byInverterInProgress].eErrorState := E_Symo_PV_Error.eSymo10TooBigValueReceived;		
							END_IF
					//Copy Data Voltage L2-L3
					rValBefWToOut := WORD_TO_REAL(arrBuffer_FC3[7]);
						lrCheckValue := rValBefWToOut * EXPT(10,WORD_TO_INT(arrBuffer_FC3[12]));	
							IF lrCheckValue >= - 3.402823E+38 AND lrCheckValue <= 3.402823E+38 THEN 
								arrVoltageL2L3[byInverterInProgress] := lrCheckValue;
							ELSE
								iStateModbus := 300;
									arrDataSymo10[byInverterInProgress].eErrorState := E_Symo_PV_Error.eSymo10TooBigValueReceived;		
							END_IF
					//Copy Data Voltage L3-L1
					rValBefWToOut := WORD_TO_REAL(arrBuffer_FC3[8]);
						lrCheckValue := rValBefWToOut * EXPT(10,WORD_TO_INT(arrBuffer_FC3[12]));	
							IF lrCheckValue >= - 3.402823E+38 AND lrCheckValue <= 3.402823E+38 THEN 
								arrVoltageL3L1[byInverterInProgress] := lrCheckValue;
							ELSE
								iStateModbus := 300;
									arrDataSymo10[byInverterInProgress].eErrorState := E_Symo_PV_Error.eSymo10TooBigValueReceived;		
							END_IF
					//Copy Data Voltage L1-N
					rValBefWToOut := WORD_TO_REAL(arrBuffer_FC3[9]);
						lrCheckValue := rValBefWToOut * EXPT(10,WORD_TO_INT(arrBuffer_FC3[12]));	
							IF lrCheckValue >= - 3.402823E+38 AND lrCheckValue <= 3.402823E+38 THEN 
								arrVoltageL1N[byInverterInProgress] := lrCheckValue;
							ELSE
								iStateModbus := 300;
									arrDataSymo10[byInverterInProgress].eErrorState := E_Symo_PV_Error.eSymo10TooBigValueReceived;		
							END_IF
					//Copy Data Voltage L2-N
					rValBefWToOut := WORD_TO_REAL(arrBuffer_FC3[10]);
						lrCheckValue := rValBefWToOut * EXPT(10,WORD_TO_INT(arrBuffer_FC3[12]));	
							IF lrCheckValue >= - 3.402823E+38 AND lrCheckValue <= 3.402823E+38 THEN 
								arrVoltageL2N[byInverterInProgress] := lrCheckValue;
							ELSE
								iStateModbus := 300;
									arrDataSymo10[byInverterInProgress].eErrorState := E_Symo_PV_Error.eSymo10TooBigValueReceived;		
							END_IF
					//Copy Data Voltage L3-N
					rValBefWToOut := WORD_TO_REAL(arrBuffer_FC3[11]);
						lrCheckValue := rValBefWToOut * EXPT(10,WORD_TO_INT(arrBuffer_FC3[12]));	
							IF lrCheckValue >= - 3.402823E+38 AND lrCheckValue <= 3.402823E+38 THEN 
								arrVoltageL3N[byInverterInProgress] := lrCheckValue;
							ELSE
								iStateModbus := 300;
									arrDataSymo10[byInverterInProgress].eErrorState := E_Symo_PV_Error.eSymo10TooBigValueReceived;		
							END_IF
					//Copy Data AC Power
					rValBefWToOut := INT_TO_REAL(WORD_TO_INT(arrBuffer_FC3[13]));
						lrCheckValue := rValBefWToOut * EXPT(10,WORD_TO_INT(arrBuffer_FC3[14]));	
							IF lrCheckValue >= - 3.402823E+38 AND lrCheckValue <= 3.402823E+38 THEN 
								arrACPower[byInverterInProgress] := lrCheckValue;
									arrDataSymo10[byInverterInProgress].lrPowerAcInverter := arrACPower[byInverterInProgress] / 1000;
							ELSE
								iStateModbus := 300;
									arrDataSymo10[byInverterInProgress].eErrorState := E_Symo_PV_Error.eSymo10TooBigValueReceived;		
							END_IF
					//Copy Data Frequency
					rValBefWToOut := WORD_TO_REAL(arrBuffer_FC3[15]);
						lrCheckValue := rValBefWToOut * EXPT(10,WORD_TO_INT(arrBuffer_FC3[16]));	
							IF lrCheckValue >= - 3.402823E+38 AND lrCheckValue <= 3.402823E+38 THEN 
								arrFrequency[byInverterInProgress] := lrCheckValue;
							ELSE
								iStateModbus := 300;
									arrDataSymo10[byInverterInProgress].eErrorState := E_Symo_PV_Error.eSymo10TooBigValueReceived;		
							END_IF
					//Copy Data Apparent Power
					rValBefWToOut := INT_TO_REAL(WORD_TO_INT(arrBuffer_FC3[17]));
						lrCheckValue := rValBefWToOut * EXPT(10,WORD_TO_INT(arrBuffer_FC3[18]));	
							IF lrCheckValue >= - 3.402823E+38 AND lrCheckValue <= 3.402823E+38 THEN 
								arrApparentPower[byInverterInProgress] := lrCheckValue;
							ELSE
								iStateModbus := 300;
									arrDataSymo10[byInverterInProgress].eErrorState := E_Symo_PV_Error.eSymo10TooBigValueReceived;		
							END_IF
					//Copy Data Reactive Power
					rValBefWToOut := INT_TO_REAL(WORD_TO_INT(arrBuffer_FC3[19]));
						lrCheckValue := rValBefWToOut * EXPT(10,WORD_TO_INT(arrBuffer_FC3[20]));	
							IF lrCheckValue >= - 3.402823E+38 AND lrCheckValue <= 3.402823E+38 THEN 
								arrReactivePower[byInverterInProgress] := lrCheckValue;
							ELSE
								iStateModbus := 300;
									arrDataSymo10[byInverterInProgress].eErrorState := E_Symo_PV_Error.eSymo10TooBigValueReceived;		
							END_IF
					//Copy Data AC production Energy
					fbConvertEnergyRegister(wInputValue_1:= arrBuffer_FC3[23], wInputValue_2:= arrBuffer_FC3[24], eByteOrderForConvert:= eByteOrder.eBigEndian, udiOutputValue=> );
					rValBefWToOut := UDINT_TO_REAL(fbConvertEnergyRegister.udiOutputValue);
						lrCheckValue := rValBefWToOut * EXPT(10,WORD_TO_INT(arrBuffer_FC3[25]));	
							IF lrCheckValue >= - 3.402823E+38 AND lrCheckValue <= 3.402823E+38 THEN 
								arrProductionEnergy[byInverterInProgress] := lrCheckValue / 1000; 
							ELSE
								iStateModbus := 300;
									arrDataSymo10[byInverterInProgress].eErrorState := E_Symo_PV_Error.eSymo10TooBigValueReceived;		
							END_IF
					//Operating State
					IF arrBuffer_FC3[37] = 1 THEN arrDataSymo10[byInverterInProgress].eOperatingStateInverter := E_Symo_PV_OperatingState.eOff;
						ELSIF arrBuffer_FC3[37] = 2 THEN arrDataSymo10[byInverterInProgress].eOperatingStateInverter := E_Symo_PV_OperatingState.eSleeping;
						ELSIF arrBuffer_FC3[37] = 3 THEN arrDataSymo10[byInverterInProgress].eOperatingStateInverter := E_Symo_PV_OperatingState.eStartingUp;
						ELSIF arrBuffer_FC3[37] = 4 THEN arrDataSymo10[byInverterInProgress].eOperatingStateInverter := E_Symo_PV_OperatingState.eTrackingPowerPoint;
						ELSIF arrBuffer_FC3[37] = 5 THEN arrDataSymo10[byInverterInProgress].eOperatingStateInverter := E_Symo_PV_OperatingState.eForcedPowerReduction;
						ELSIF arrBuffer_FC3[37] = 6 THEN arrDataSymo10[byInverterInProgress].eOperatingStateInverter := E_Symo_PV_OperatingState.eShuttingDown;
						ELSIF arrBuffer_FC3[37] = 7 THEN arrDataSymo10[byInverterInProgress].eOperatingStateInverter := E_Symo_PV_OperatingState.eFaults;
						ELSIF arrBuffer_FC3[37] = 8 THEN arrDataSymo10[byInverterInProgress].eOperatingStateInverter := E_Symo_PV_OperatingState.eStandby;
						ELSE arrDataSymo10[byInverterInProgress].eOperatingStateInverter := E_Symo_PV_OperatingState.eNoDataReceived;
					END_IF
					//Next Step
					IF iStateModbus = 2 THEN
						fbMBRead_FC3.bExecute := FALSE;
							timDelay.IN := FALSE;
								iStateModbus := 3;
									arrDataSymo10[byInverterInProgress].bError := FALSE; 
										arrDataSymo10[byInverterInProgress].eErrorState := E_Symo_PV_Error.eNoError;
					END_IF
		END_IF
			
		//Error from Inverter
		IF NOT fbMBRead_FC3.bBusy AND NOT fbMBRead_FC3.bError AND timDelay.Q AND arrDataSymo10[byInverterInProgress].eOperatingStateInverter = E_Symo_PV_OperatingState.eFaults THEN
			iStateModbus := 300;
				arrDataSymo10[byInverterInProgress].eErrorState := E_Symo_PV_Error.eSymo10Error;
		END_IF
		
		//Error about scalling factor
		IF (NOT fbMBRead_FC3.bBusy AND NOT fbMBRead_FC3.bError AND timDelay.Q AND (WORD_TO_INT(arrBuffer_FC3[5]) < -10 OR WORD_TO_INT(arrBuffer_FC3[5]) > 10 OR WORD_TO_INT(arrBuffer_FC3[12]) < -10 OR WORD_TO_INT(arrBuffer_FC3[12]) > 10 OR
			WORD_TO_INT(arrBuffer_FC3[14]) < -10 OR WORD_TO_INT(arrBuffer_FC3[14]) > 10 OR WORD_TO_INT(arrBuffer_FC3[16]) < -10 OR WORD_TO_INT(arrBuffer_FC3[16]) > 10 OR WORD_TO_INT(arrBuffer_FC3[18]) < -10 OR WORD_TO_INT(arrBuffer_FC3[18]) > 10 OR
				WORD_TO_INT(arrBuffer_FC3[20]) < -10 OR WORD_TO_INT(arrBuffer_FC3[20]) > 10 OR WORD_TO_INT(arrBuffer_FC3[25]) < -10 OR WORD_TO_INT(arrBuffer_FC3[25]) > 10)) THEN
					iStateModbus := 300;
						arrDataSymo10[byInverterInProgress].eErrorState := E_Symo_PV_Error.eSymo10TooBigValueReceived;
		END_IF
	 
		//Error or Timeout
		IF FPError_FC_3.Q OR timTimeout.Q THEN
			iStateModbus := 300;
				arrDataSymo10[byInverterInProgress].eErrorState := E_Symo_PV_Error.eModbusTCPError;
		END_IF

	3://Calculate the sum of the values
		iStateModbus_CP := iStateModbus;
		
		lrCounterEnergyProduction := 0;
			fbElMeter.lrCurrentL1 := 0;
		fbElMeter.lrCurrentL2 := 0;	
			fbElMeter.lrCurrentL3 := 0;
		fbElMeter.lrVoltageL1N := 0;
			fbElMeter.lrVoltageL2N := 0;
		fbElMeter.lrVoltageL3N := 0;
			fbElMeter.lrVoltageL1L2 := 0;
		fbElMeter.lrVoltageL2L3 := 0;
			fbElMeter.lrVoltageL3L1 := 0;
		fbElMeter.lrPowerTotal := 0;
			fbElMeter.lrFrequency := 0;
		fbElMeter.lrReactivePowerTotal := 0;
			fbElMeter.lrApparentPowerTotal := 0;
		
		FOR byLPForInverter := 1 TO 30 BY 1 DO 
			lrCounterEnergyProduction := lrCounterEnergyProduction + arrProductionEnergy[byLPForInverter];
			IF lrCounterEnergyProduction > fbElMeter.lrCounterEnergyT1_Production THEN
				fbElMeter.lrCounterEnergyT1_Production := lrCounterEnergyProduction;
			END_IF
				fbElMeter.lrCurrentL1 := fbElMeter.lrCurrentL1 + arrCurrentL1[byLPForInverter];
			fbElMeter.lrCurrentL2 := fbElMeter.lrCurrentL2 + arrCurrentL2[byLPForInverter];	
				fbElMeter.lrCurrentL3 := fbElMeter.lrCurrentL3 + arrCurrentL3[byLPForInverter];
			IF byTotalInverter > 0 THEN
				fbElMeter.lrVoltageL1N := (fbElMeter.lrVoltageL1N + arrVoltageL1N[byLPForInverter]) / byTotalInverter;
					fbElMeter.lrVoltageL2N := (fbElMeter.lrVoltageL2N + arrVoltageL2N[byLPForInverter]) / byTotalInverter;
				fbElMeter.lrVoltageL3N := (fbElMeter.lrVoltageL3N + arrVoltageL3N[byLPForInverter]) / byTotalInverter;
					fbElMeter.lrVoltageL1L2 := (fbElMeter.lrVoltageL1L2 + arrVoltageL1L2[byLPForInverter]) / byTotalInverter;
				fbElMeter.lrVoltageL2L3 := (fbElMeter.lrVoltageL2L3 + arrVoltageL2L3[byLPForInverter]) / byTotalInverter;
					fbElMeter.lrVoltageL3L1 := (fbElMeter.lrVoltageL3L1 + arrVoltageL3L1[byLPForInverter]) / byTotalInverter;
				fbElMeter.lrFrequency := (fbElMeter.lrFrequency + arrFrequency[byLPForInverter]) / byTotalInverter;
			END_IF
					fbElMeter.lrPowerTotal := fbElMeter.lrPowerTotal + arrACPower[byLPForInverter];
				fbElMeter.lrReactivePowerTotal := fbElMeter.lrReactivePowerTotal + arrReactivePower[byLPForInverter];
					fbElMeter.lrApparentPowerTotal := fbElMeter.lrApparentPowerTotal + arrApparentPower[byLPForInverter];
		END_FOR	
					
		fbElMeter.lrTotalCounterEnergy_Production := fbElMeter.lrCounterEnergyT1_Production; 
		
			iStateModbus := 1;
				
	300://Error
		iStateModbus_CP := iStateModbus;
			timDelay.IN := FALSE;
				fbMBRead_FC3.bExecute := FALSE;
					arrDataSymo10[byInverterInProgress].bError := TRUE;
						iStateModbus := 1;				
							
END_CASE

(*------------------------------------------------------------------------------------------Modbus TCP Function---------------------------------------------------------------------------------------------*)

fbMBRead_FC3(sIPAddr:= sIPAdress, nTCPPort:= 502, cbLength:= SIZEOF(arrBuffer_FC3), pDestAddr:= ADR(arrBuffer_FC3), tTimeout:= T#10S );
	FPError_FC_3(CLK:= fbMBRead_FC3.bError, Q=> );

(*----------------------------------------------------------------------------------------Electric Meter Data----------------------------------------------------------------------------------------------*)

//Error and Warning
bErrorDevice := FALSE;
	FOR byLPForInverter := 1 TO 30 BY 1 DO
		IF arrDataSymo10[byLPForInverter].bError THEN bErrorDevice := TRUE; END_IF 
	END_FOR 

IF timDissableFunctions.Q THEN fbElMeter.bWarning := TRUE; fbElMeter.iWarningCode := 0; ELSE fbElMeter.bWarning := FALSE; END_IF   
	IF bErrorDevice OR Lynus_Standards.GVL_Energy.stNumberOfDevices.diNumberOfElectricMeters > Constants_Energy.diMaxNumberOfElectricMeters THEN fbElMeter.bError := TRUE; ELSE fbElMeter.bError := FALSE; END_IF  

IF Lynus_Standards.GVL_Energy.stNumberOfDevices.diNumberOfElectricMeters > Constants_Energy.diMaxNumberOfElectricMeters THEN fbElMeter.iErrorCode := 1;
ELSIF bErrorDevice THEN fbElMeter.iErrorCode := 0;
END_IF  

//Read Out Data done for EM Function
IF iStateModbus <> 3 THEN fbElMeter.bReadOutDataDone := TRUE; ELSE fbElMeter.bReadOutDataDone := FALSE; END_IF

//Function block for meter data
fbElMeter(
	bEnable:= bEnable AND NOT timDissableFunctions.Q, 
	bError:= , 
	bEnableReadOutFunction:= FALSE, 
	bWriteWithDelay:= TRUE,
	bPowerDataInvers:= TRUE, 
	bReadOutDataDone:= ,
	iTimeReadOutInterval:= , 
	iErrorCode:= , 
	iWarningCode:= , 
	lrTotalCounterEnergy_Consumption:= 0, 
	lrTotalCounterEnergy_Production:= , 
	lrCounterEnergyT1_Consumption:= 0, 
	lrCounterEnergyT2_Consumption:= 0, 
	lrCounterEnergyT1_Production:= , 
	lrCounterEnergyT2_Production:= 0, 
	lrCurrentL1:= , 
	lrVoltageL1N:= , 
	lrVoltageL1L2:= , 
	lrPowerL1:= 0, 
	lrCurrentL2:= , 
	lrVoltageL2N:= , 
	lrVoltageL2L3:= , 
	lrPowerL2:= 0, 
	lrCurrentL3:= , 
	lrVoltageL3N:= , 
	lrVoltageL3L1:= , 
	lrPowerL3:= 0, 
	lrPowerTotal:= , 
	lrFrequency:= , 
	lrReactivePowerTotal:= , 
	lrApparentPowerTotal:= , 
	tTimDelayOutput:= T#5S, 
	stDataEMOutPower=> , 
	stDataEMOutPowerDelay=> stDataEMPower_PV, 
	stDataEMOutCounter=> ,
	stDataEMOutCounterDelay=> stDataEMCounter_PV, 
	bReadOutMeter=> );

(*-----------------------------------------------------------Handle data to Global structure for the Electric Meter system-----------------------------------------------------------------*)

CASE iStateGVLData OF
	
	0://Init Step
		byWaitInStep := 0;
			diCounterForGVL := 1;
	
	1://Wait for 4 Steps before clean al Data on GVL
		byWaitInStep := byWaitInStep + 1;
			IF byWaitInStep >= 4 AND fbNumberDevice.bNumberIsCalculatet THEN iStateGVLData := 2; END_IF
				//To much Devices, back to the Init step
				IF byWaitInStep >= 4 AND NOT fbNumberDevice.bNumberIsCalculatet THEN iStateGVLData := 0; END_IF	
			
	2://Clear all Data in GVL
		Lynus_Standards.GVL_Energy.stDataElectricMeters[diCounterForGVL].bEnabled := FALSE;	
			Lynus_Standards.GVL_Energy.stDataElectricMeters[diCounterForGVL].byErrorWarning := 0;
				Lynus_Standards.GVL_Energy.stDataElectricMeters[diCounterForGVL].lrCounterEnergyT1_Consumption := 0;
					Lynus_Standards.GVL_Energy.stDataElectricMeters[diCounterForGVL].lrCounterEnergyT1_Production := 0;
						Lynus_Standards.GVL_Energy.stDataElectricMeters[diCounterForGVL].lrCounterEnergyT2_Consumption := 0;
							Lynus_Standards.GVL_Energy.stDataElectricMeters[diCounterForGVL].lrCounterEnergyT2_Production := 0;
								Lynus_Standards.GVL_Energy.stDataElectricMeters[diCounterForGVL].lrPower := 0;
									Lynus_Standards.GVL_Energy.stDataElectricMeters[diCounterForGVL].lrPowerConsumption := 0;
										Lynus_Standards.GVL_Energy.stDataElectricMeters[diCounterForGVL].lrPowerConsumption := 0;
											Lynus_Standards.GVL_Energy.stDataElectricMeters[diCounterForGVL].lrPowerProduction := 0;
												Lynus_Standards.GVL_Energy.stDataElectricMeters[diCounterForGVL].lrTotalCounterEnergy_Consumption := 0;
													Lynus_Standards.GVL_Energy.stDataElectricMeters[diCounterForGVL].lrTotalCounterEnergy_Production := 0;
		
		diCounterForGVL := diCounterForGVL + 1;
			diCounterForGVL := LIMIT(0,diCounterForGVL,Constants_Energy.diMaxNumberOfElectricMeters);
				//Back to the init step
				IF diCounterForGVL >= Constants_Energy.diMaxNumberOfElectricMeters THEN iStateGVLData := 0; END_IF

END_CASE 	 

IF diNrOfEM_OUT_PV > 0 AND fbNumberDevice.bNumberIsCalculatet THEN
	Lynus_Standards.GVL_Energy.stDataElectricMeters[diNrOfEM_OUT_PV].bEnabled := fbElMeter.stDataEMOutPower.bEnabled;
		Lynus_Standards.GVL_Energy.stDataElectricMeters[diNrOfEM_OUT_PV].byErrorWarning := fbElMeter.stDataEMOutPower.byErrorWarning;
			Lynus_Standards.GVL_Energy.stDataElectricMeters[diNrOfEM_OUT_PV].lrCounterEnergyT1_Consumption := fbElMeter.stDataEMOutCounter.lrCounterEnergyT1_Consumption;
				Lynus_Standards.GVL_Energy.stDataElectricMeters[diNrOfEM_OUT_PV].lrCounterEnergyT1_Production := fbElMeter.stDataEMOutCounter.lrCounterEnergyT1_Production;
					Lynus_Standards.GVL_Energy.stDataElectricMeters[diNrOfEM_OUT_PV].lrCounterEnergyT2_Consumption := fbElMeter.stDataEMOutCounter.lrCounterEnergyT2_Consumption;
						Lynus_Standards.GVL_Energy.stDataElectricMeters[diNrOfEM_OUT_PV].lrCounterEnergyT2_Production := fbElMeter.stDataEMOutCounter.lrCounterEnergyT2_Production;		
							Lynus_Standards.GVL_Energy.stDataElectricMeters[diNrOfEM_OUT_PV].lrPower := fbElMeter.stDataEMOutPower.lrPowerTotal;
								Lynus_Standards.GVL_Energy.stDataElectricMeters[diNrOfEM_OUT_PV].lrPowerConsumption := fbElMeter.stDataEMOutPower.lrPowerConsumption;
									Lynus_Standards.GVL_Energy.stDataElectricMeters[diNrOfEM_OUT_PV].lrPowerProduction := fbElMeter.stDataEMOutPower.lrPowerProduction;
										Lynus_Standards.GVL_Energy.stDataElectricMeters[diNrOfEM_OUT_PV].lrTotalCounterEnergy_Consumption := fbElMeter.stDataEMOutCounter.lrTotalCounterEnergy_Consumption;
											Lynus_Standards.GVL_Energy.stDataElectricMeters[diNrOfEM_OUT_PV].lrTotalCounterEnergy_Production := fbElMeter.stDataEMOutCounter.lrTotalCounterEnergy_Production;
END_IF

(*----------------------------------------------------------Save persistent data----------------------------------------------------------------*)

arrPD[1](lrValue:= BOOL_TO_LREAL(bEnable), bEventBasedActive=> );
arrPD[2](lrValue:= BYTE_TO_LREAL(arrUnitID_Inverter[1]), bEventBasedActive=> );
arrPD[3](lrValue:= BYTE_TO_LREAL(arrUnitID_Inverter[2]), bEventBasedActive=> );
arrPD[4](lrValue:= BYTE_TO_LREAL(arrUnitID_Inverter[3]), bEventBasedActive=> );
arrPD[5](lrValue:= BYTE_TO_LREAL(arrUnitID_Inverter[4]), bEventBasedActive=> );
arrPD[6](lrValue:= BYTE_TO_LREAL(arrUnitID_Inverter[5]), bEventBasedActive=> );
arrPD[7](lrValue:= BYTE_TO_LREAL(arrUnitID_Inverter[6]), bEventBasedActive=> );
arrPD[8](lrValue:= BYTE_TO_LREAL(arrUnitID_Inverter[7]), bEventBasedActive=> );
arrPD[9](lrValue:= BYTE_TO_LREAL(arrUnitID_Inverter[8]), bEventBasedActive=> );
arrPD[10](lrValue:= BYTE_TO_LREAL(arrUnitID_Inverter[9]), bEventBasedActive=> );
arrPD[11](lrValue:= BYTE_TO_LREAL(arrUnitID_Inverter[10]), bEventBasedActive=> );
arrPD[12](lrValue:= BYTE_TO_LREAL(arrUnitID_Inverter[11]), bEventBasedActive=> );
arrPD[13](lrValue:= BYTE_TO_LREAL(arrUnitID_Inverter[12]), bEventBasedActive=> );
arrPD[14](lrValue:= BYTE_TO_LREAL(arrUnitID_Inverter[13]), bEventBasedActive=> );
arrPD[15](lrValue:= BYTE_TO_LREAL(arrUnitID_Inverter[14]), bEventBasedActive=> );
arrPD[16](lrValue:= BYTE_TO_LREAL(arrUnitID_Inverter[15]), bEventBasedActive=> );
arrPD[17](lrValue:= BYTE_TO_LREAL(arrUnitID_Inverter[16]), bEventBasedActive=> );
arrPD[18](lrValue:= BYTE_TO_LREAL(arrUnitID_Inverter[17]), bEventBasedActive=> );
arrPD[19](lrValue:= BYTE_TO_LREAL(arrUnitID_Inverter[18]), bEventBasedActive=> );
arrPD[20](lrValue:= BYTE_TO_LREAL(arrUnitID_Inverter[19]), bEventBasedActive=> );
arrPD[21](lrValue:= BYTE_TO_LREAL(arrUnitID_Inverter[20]), bEventBasedActive=> );
arrPD[22](lrValue:= BYTE_TO_LREAL(arrUnitID_Inverter[21]), bEventBasedActive=> );
arrPD[23](lrValue:= BYTE_TO_LREAL(arrUnitID_Inverter[22]), bEventBasedActive=> );
arrPD[24](lrValue:= BYTE_TO_LREAL(arrUnitID_Inverter[23]), bEventBasedActive=> );
arrPD[25](lrValue:= BYTE_TO_LREAL(arrUnitID_Inverter[24]), bEventBasedActive=> );
arrPD[26](lrValue:= BYTE_TO_LREAL(arrUnitID_Inverter[25]), bEventBasedActive=> );
arrPD[27](lrValue:= BYTE_TO_LREAL(arrUnitID_Inverter[26]), bEventBasedActive=> );
arrPD[28](lrValue:= BYTE_TO_LREAL(arrUnitID_Inverter[27]), bEventBasedActive=> );
arrPD[29](lrValue:= BYTE_TO_LREAL(arrUnitID_Inverter[28]), bEventBasedActive=> );
arrPD[30](lrValue:= BYTE_TO_LREAL(arrUnitID_Inverter[29]), bEventBasedActive=> );
arrPD[31](lrValue:= BYTE_TO_LREAL(arrUnitID_Inverter[30]), bEventBasedActive=> );
PD_String(sText:= sIPAdress, bEventBasedActive=> );

END_FUNCTION_BLOCK

// ---- POUs/prgCS.TcPOU
PROGRAM prgCS
VAR
	fb_CS1 :	fb_ECS_KEBA_P30_noWrite;	
	fb_CS2 :	fb_ECS_KEBA_P30_noWrite;	
	fb_CS3 :	fb_ECS_KEBA_P30_noWrite;	
	fb_CS4 :	fb_ECS_KEBA_P30_noWrite;
	fb_CS5 :	fb_ECS_KEBA_P30_noWrite;	
	fb_CS6 :	fb_ECS_KEBA_P30_noWrite;
	fb_CS7 :	fb_ECS_KEBA_P30_noWrite;	
	fb_CS8 :	fb_ECS_KEBA_P30_noWrite;
	fb_CS9 :	fb_ECS_KEBA_P30_noWrite;	
	fb_CS10 :	fb_ECS_KEBA_P30_noWrite;

	lr_Power_CS1			: LREAL;						//{#lynus.ag#()}
	lr_EnergyTotal_CS1		: LREAL;						//{#lynus.ag#()}
	bool_CarConnected_CS1	: BOOL;							//{#lynus.ag#()}
	lr_Power_CS2			: LREAL;						//{#lynus.ag#()}
	lr_EnergyTotal_CS2		: LREAL;						//{#lynus.ag#()}
	bool_CarConnected_CS2	: BOOL;							//{#lynus.ag#()}
	lr_Power_CS3			: LREAL;						//{#lynus.ag#()}
	lr_EnergyTotal_CS3		: LREAL;						//{#lynus.ag#()}
	bool_CarConnected_CS3	: BOOL;							//{#lynus.ag#()}
	lr_Power_CS4			: LREAL;						//{#lynus.ag#()}
	lr_EnergyTotal_CS4		: LREAL;						//{#lynus.ag#()}
	bool_CarConnected_CS4	: BOOL;							//{#lynus.ag#()}
	lr_Power_CS5			: LREAL;						//{#lynus.ag#()}
	lr_EnergyTotal_CS5		: LREAL;						//{#lynus.ag#()}
	bool_CarConnected_CS5	: BOOL;							//{#lynus.ag#()}
	lr_Power_CS6			: LREAL;						//{#lynus.ag#()}
	lr_EnergyTotal_CS6		: LREAL;						//{#lynus.ag#()}
	bool_CarConnected_CS6	: BOOL;							//{#lynus.ag#()}
	lr_Power_CS7			: LREAL;						//{#lynus.ag#()}
	lr_EnergyTotal_CS7		: LREAL;						//{#lynus.ag#()}
	bool_CarConnected_CS7	: BOOL;							//{#lynus.ag#()}
	lr_Power_CS8			: LREAL;						//{#lynus.ag#()}
	lr_EnergyTotal_CS8		: LREAL;						//{#lynus.ag#()}
	bool_CarConnected_CS8	: BOOL;							//{#lynus.ag#()}
	lr_Power_CS9			: LREAL;						//{#lynus.ag#()}
	lr_EnergyTotal_CS9		: LREAL;						//{#lynus.ag#()}
	bool_CarConnected_CS9	: BOOL;							//{#lynus.ag#()}
	lr_Power_CS10			: LREAL;						//{#lynus.ag#()}
	lr_EnergyTotal_CS10		: LREAL;						//{#lynus.ag#()}
	bool_CarConnected_CS10	: BOOL;							//{#lynus.ag#()}
	lr_Power_CS_total		: LREAL;						//{#lynus.ag#()}
	usint_CarConnected_CS1	: USINT;						//{#lynus.ag#()}
	usint_CarConnected_CS2	: USINT;						//{#lynus.ag#()}
	usint_CarConnected_CS3	: USINT;						//{#lynus.ag#()}
	usint_CarConnected_CS4	: USINT;						//{#lynus.ag#()}
	usint_CarConnected_CS5	: USINT;						//{#lynus.ag#()}
	usint_CarConnected_CS6	: USINT;						//{#lynus.ag#()}
	usint_CarConnected_CS7	: USINT;						//{#lynus.ag#()}
	usint_CarConnected_CS8	: USINT;						//{#lynus.ag#()}
	usint_CarConnected_CS9	: USINT;						//{#lynus.ag#()}
	usint_CarConnected_CS10	: USINT;						//{#lynus.ag#()}
	r_ChargeTime_CS1		: REAL;							//{#lynus.ag#()}
	r_ChargeTime_CS2		: REAL;							//{#lynus.ag#()}
	r_ChargeTime_CS3		: REAL;							//{#lynus.ag#()}
	r_ChargeTime_CS4		: REAL;							//{#lynus.ag#()}
	r_ChargeTime_CS5		: REAL;							//{#lynus.ag#()}
	r_ChargeTime_CS6		: REAL;							//{#lynus.ag#()}
	r_ChargeTime_CS7		: REAL;							//{#lynus.ag#()}
	r_ChargeTime_CS8		: REAL;							//{#lynus.ag#()}
	r_ChargeTime_CS9		: REAL;							//{#lynus.ag#()}
	r_ChargeTime_CS10		: REAL;							//{#lynus.ag#()}
	lr_EnergySession_CS1	: LREAL;						//{#lynus.ag#()}
	lr_EnergySession_CS2	: LREAL;						//{#lynus.ag#()}
	lr_EnergySession_CS3	: LREAL;						//{#lynus.ag#()}
	lr_EnergySession_CS4	: LREAL;						//{#lynus.ag#()}
	lr_EnergySession_CS5	: LREAL;						//{#lynus.ag#()}
	lr_EnergySession_CS6	: LREAL;						//{#lynus.ag#()}
	lr_EnergySession_CS7	: LREAL;						//{#lynus.ag#()}
	lr_EnergySession_CS8	: LREAL;						//{#lynus.ag#()}
	lr_EnergySession_CS9	: LREAL;						//{#lynus.ag#()}
	lr_EnergySession_CS10	: LREAL;						//{#lynus.ag#()}


END_VAR

fb_CS1(
	bEnable:= TRUE, 
	bEnable_write := FALSE,
	bPowerDataInvers:= , 
	byElectricFuseLine:= , 
	uiFailsafeCurrent:= , 
	uiFailsafeTimeOut:= , 
	diNrOfEMS_IN:= , 
	diNrOfEM_IN_CS:= , 
	sIPAdress:= '10.30.140.1', 
	stSetupECS:= , 
	stDataECS=> , 
	diNrOfECS_OUT=> , 
	lrTotalPowerECSRealTime=> );
lr_Power_CS1 			:= fb_CS1.stDataECS.lrTotalPower;
lr_EnergyTotal_CS1		:= fb_CS1.stDataECS.lrCounterEnergyT1_Consumption/10;
bool_CarConnected_CS1	:= fb_CS1.stDataECS.bCarConnected;
r_ChargeTime_CS1		:= fb_CS1.stDataECS.arrChargingTimeInMin[1];
lr_EnergySession_CS1	:= fb_CS1.stDataECS.arrSocketEnergySession[1]/10;

fb_CS2(
	bEnable:= TRUE, 
	bEnable_write := FALSE,
	bPowerDataInvers:= , 
	byElectricFuseLine:= , 
	uiFailsafeCurrent:= , 
	uiFailsafeTimeOut:= , 
	diNrOfEMS_IN:= , 
	diNrOfEM_IN_CS:= , 
	sIPAdress:= '10.30.140.2', 
	stSetupECS:= , 
	stDataECS=> , 
	diNrOfECS_OUT=> , 
	lrTotalPowerECSRealTime=> );
lr_Power_CS2 			:= fb_CS2.stDataECS.lrTotalPower;
lr_EnergyTotal_CS2		:= fb_CS2.stDataECS.lrCounterEnergyT1_Consumption/10;
bool_CarConnected_CS2	:= fb_CS2.stDataECS.bCarConnected;
r_ChargeTime_CS2		:= fb_CS2.stDataECS.arrChargingTimeInMin[1];
lr_EnergySession_CS2	:= fb_CS2.stDataECS.arrSocketEnergySession[1]/10;
	
fb_CS3(
	bEnable:= TRUE, 
	bEnable_write := FALSE,
	bPowerDataInvers:= , 
	byElectricFuseLine:= , 
	uiFailsafeCurrent:= , 
	uiFailsafeTimeOut:= , 
	diNrOfEMS_IN:= , 
	diNrOfEM_IN_CS:= , 
	sIPAdress:= '10.30.140.3', 
	stSetupECS:= , 
	stDataECS=> , 
	diNrOfECS_OUT=> , 
	lrTotalPowerECSRealTime=> );
lr_Power_CS3 			:= fb_CS3.stDataECS.lrTotalPower;
lr_EnergyTotal_CS3		:= fb_CS3.stDataECS.lrCounterEnergyT1_Consumption/10;
bool_CarConnected_CS3	:= fb_CS3.stDataECS.bCarConnected;
r_ChargeTime_CS3		:= fb_CS3.stDataECS.arrChargingTimeInMin[1];
lr_EnergySession_CS3	:= fb_CS3.stDataECS.arrSocketEnergySession[1]/10;
	
fb_CS4(
	bEnable:= TRUE, 
	bEnable_write := FALSE,
	bPowerDataInvers:= , 
	byElectricFuseLine:= , 
	uiFailsafeCurrent:= , 
	uiFailsafeTimeOut:= , 
	diNrOfEMS_IN:= , 
	diNrOfEM_IN_CS:= , 
	sIPAdress:= '10.30.140.4', 
	stSetupECS:= , 
	stDataECS=> , 
	diNrOfECS_OUT=> , 
	lrTotalPowerECSRealTime=> );
lr_Power_CS4 			:= fb_CS4.stDataECS.lrTotalPower;
lr_EnergyTotal_CS4		:= fb_CS4.stDataECS.lrCounterEnergyT1_Consumption/10;
bool_CarConnected_CS4	:= fb_CS4.stDataECS.bCarConnected;
r_ChargeTime_CS4		:= fb_CS4.stDataECS.arrChargingTimeInMin[1];
lr_EnergySession_CS4	:= fb_CS4.stDataECS.arrSocketEnergySession[1]/10;
	
fb_CS5(
	bEnable:= TRUE, 
	bEnable_write := FALSE,
	bPowerDataInvers:= , 
	byElectricFuseLine:= , 
	uiFailsafeCurrent:= , 
	uiFailsafeTimeOut:= , 
	diNrOfEMS_IN:= , 
	diNrOfEM_IN_CS:= , 
	sIPAdress:= '10.30.140.5', 
	stSetupECS:= , 
	stDataECS=> , 
	diNrOfECS_OUT=> , 
	lrTotalPowerECSRealTime=> );
lr_Power_CS5 			:= fb_CS5.stDataECS.lrTotalPower;
lr_EnergyTotal_CS5		:= fb_CS5.stDataECS.lrCounterEnergyT1_Consumption/10;
bool_CarConnected_CS5	:= fb_CS5.stDataECS.bCarConnected;
r_ChargeTime_CS5		:= fb_CS5.stDataECS.arrChargingTimeInMin[1];
lr_EnergySession_CS5	:= fb_CS5.stDataECS.arrSocketEnergySession[1]/10;

fb_CS6(
	bEnable:= TRUE, 
	bEnable_write := FALSE,
	bPowerDataInvers:= , 
	byElectricFuseLine:= , 
	uiFailsafeCurrent:= , 
	uiFailsafeTimeOut:= , 
	diNrOfEMS_IN:= , 
	diNrOfEM_IN_CS:= , 
	sIPAdress:= '10.30.140.6', 
	stSetupECS:= , 
	stDataECS=> , 
	diNrOfECS_OUT=> , 
	lrTotalPowerECSRealTime=> );
lr_Power_CS6 			:= fb_CS6.stDataECS.lrTotalPower;
lr_EnergyTotal_CS6		:= fb_CS6.stDataECS.lrCounterEnergyT1_Consumption/10;
bool_CarConnected_CS6	:= fb_CS6.stDataECS.bCarConnected;
r_ChargeTime_CS6		:= fb_CS6.stDataECS.arrChargingTimeInMin[1];
lr_EnergySession_CS6   	:= fb_CS6.stDataECS.arrSocketEnergySession[1]/10;

fb_CS7(
	bEnable:= TRUE, 
	bEnable_write := FALSE,
	bPowerDataInvers:= , 
	byElectricFuseLine:= , 
	uiFailsafeCurrent:= , 
	uiFailsafeTimeOut:= , 
	diNrOfEMS_IN:= , 
	diNrOfEM_IN_CS:= , 
	sIPAdress:= '10.30.140.7', 
	stSetupECS:= , 
	stDataECS=> , 
	diNrOfECS_OUT=> , 
	lrTotalPowerECSRealTime=> );
lr_Power_CS7			:= fb_CS7.stDataECS.lrTotalPower;
lr_EnergyTotal_CS7		:= fb_CS7.stDataECS.lrCounterEnergyT1_Consumption/10;
bool_CarConnected_CS7	:= fb_CS7.stDataECS.bCarConnected;
r_ChargeTime_CS7		:= fb_CS7.stDataECS.arrChargingTimeInMin[1];
lr_EnergySession_CS7	:= fb_CS7.stDataECS.arrSocketEnergySession[1]/10;

fb_CS8(
	bEnable:= TRUE, 
	bEnable_write := FALSE,
	bPowerDataInvers:= , 
	byElectricFuseLine:= , 
	uiFailsafeCurrent:= , 
	uiFailsafeTimeOut:= , 
	diNrOfEMS_IN:= , 
	diNrOfEM_IN_CS:= , 
	sIPAdress:= '10.30.140.8', 
	stSetupECS:= , 
	stDataECS=> , 
	diNrOfECS_OUT=> , 
	lrTotalPowerECSRealTime=> );
lr_Power_CS8 			:= fb_CS8.stDataECS.lrTotalPower;
lr_EnergyTotal_CS8		:= fb_CS8.stDataECS.lrCounterEnergyT1_Consumption/10;
bool_CarConnected_CS8	:= fb_CS8.stDataECS.bCarConnected;
r_ChargeTime_CS8		:= fb_CS8.stDataECS.arrChargingTimeInMin[1];
lr_EnergySession_CS8	:= fb_CS8.stDataECS.arrSocketEnergySession[1]/10;

fb_CS9(
	bEnable:= TRUE, 
	bEnable_write := FALSE,
	bPowerDataInvers:= , 
	byElectricFuseLine:= , 
	uiFailsafeCurrent:= , 
	uiFailsafeTimeOut:= , 
	diNrOfEMS_IN:= , 
	diNrOfEM_IN_CS:= , 
	sIPAdress:= '10.30.140.9', 
	stSetupECS:= , 
	stDataECS=> , 
	diNrOfECS_OUT=> , 
	lrTotalPowerECSRealTime=> );
lr_Power_CS9 			:= fb_CS9.stDataECS.lrTotalPower;
lr_EnergyTotal_CS9		:= fb_CS9.stDataECS.lrCounterEnergyT1_Consumption/10;
bool_CarConnected_CS9	:= fb_CS9.stDataECS.bCarConnected;
r_ChargeTime_CS9		:= fb_CS9.stDataECS.arrChargingTimeInMin[1];
lr_EnergySession_CS9	:= fb_CS9.stDataECS.arrSocketEnergySession[1]/10;

fb_CS10(
	bEnable:= TRUE, 
	bEnable_write := FALSE,
	bPowerDataInvers:= , 
	byElectricFuseLine:= , 
	uiFailsafeCurrent:= , 
	uiFailsafeTimeOut:= , 
	diNrOfEMS_IN:= , 
	diNrOfEM_IN_CS:= , 
	sIPAdress:= '10.30.140.10', 
	stSetupECS:= , 
	stDataECS=> , 
	diNrOfECS_OUT=> , 
	lrTotalPowerECSRealTime=> );
lr_Power_CS10 			:= fb_CS10.stDataECS.lrTotalPower;
lr_EnergyTotal_CS10		:= fb_CS10.stDataECS.lrCounterEnergyT1_Consumption/10;
bool_CarConnected_CS10	:= fb_CS10.stDataECS.bCarConnected;
r_ChargeTime_CS10		:= fb_CS10.stDataECS.arrChargingTimeInMin[1];
lr_EnergySession_CS10	:= fb_CS10.stDataECS.arrSocketEnergySession[1]/10;


lr_Power_CS_total := lr_Power_CS1 + lr_Power_CS2 + lr_Power_CS3 + lr_Power_CS4 + lr_Power_CS5 + lr_Power_CS6 + lr_Power_CS7 + lr_Power_CS8 + lr_Power_CS9 + lr_Power_CS10;


IF bool_CarConnected_CS1 THEN 
	usint_CarConnected_CS1 := 251;
ELSE
	usint_CarConnected_CS1 := 0;
END_IF
IF bool_CarConnected_CS2 THEN 
	usint_CarConnected_CS2 := 251;
ELSE
	usint_CarConnected_CS2 := 0;
END_IF
IF bool_CarConnected_CS3 THEN 
	usint_CarConnected_CS3 := 251;
ELSE
	usint_CarConnected_CS3 := 0;
END_IF
IF bool_CarConnected_CS4 THEN 
	usint_CarConnected_CS4 := 251;
ELSE
	usint_CarConnected_CS4 := 0;
END_IF
IF bool_CarConnected_CS5 THEN 
	usint_CarConnected_CS5 := 251;
ELSE
	usint_CarConnected_CS5 := 0;
END_IF
IF bool_CarConnected_CS6 THEN 
	usint_CarConnected_CS6 := 251;
ELSE
	usint_CarConnected_CS6 := 0;
END_IF
IF bool_CarConnected_CS7 THEN 
	usint_CarConnected_CS7 := 251;
ELSE
	usint_CarConnected_CS7 := 0;
END_IF
IF bool_CarConnected_CS8 THEN 
	usint_CarConnected_CS8 := 251;
ELSE
	usint_CarConnected_CS8 := 0;
END_IF
IF bool_CarConnected_CS9 THEN 
	usint_CarConnected_CS9 := 251;
ELSE
	usint_CarConnected_CS9 := 0;
END_IF
IF bool_CarConnected_CS10 THEN 
	usint_CarConnected_CS10 := 251;
ELSE
	usint_CarConnected_CS10 := 0;
END_IF

END_PROGRAM

